// TIA Portal V15.1 export
// export: Created 2024-06-21T08:41:18.6949066Z, ExportSetting WithDefaults, DisplayName Totally Integrated Automation Portal, DisplayVersion V15.1 Update 5, DisplayName TIA Portal Openness, DisplayVersion V15.1 Update 5, DisplayName SINAMICS Startdrive Advanced, DisplayVersion V15.1, DisplayName G130, G150, S120, S150, SINAMICS MV, S210, DisplayVersion V15.1, DisplayName G110M, G120, G120C, G120D, G120P, DisplayVersion V15.1, DisplayName STEP 7 Professional, DisplayVersion V15.1 Update 5, DisplayName STEP 7 Safety, DisplayVersion V15.1, DisplayName WinCC Professional, DisplayVersion V15.1 Update 5, DisplayName SIMATIC Visualization Architect, DisplayVersion V15.1
FUNCTION_BLOCK "LGBLineConv-MDXPN-DFS22B"   // FB6682, FBD
TITLE = LGBLineConv-MDXPN-DFS22B
{ S7_Optimized_Access := 'TRUE' }
VERSION : 0.1
// stored: AutoNumber false, IsIECCheckEnabled false, IsRetainMemResEnabled false, MemoryReserve 100, SetENOAutomatically False, UDAEnableTagReadback false
   VAR_INPUT
      I_DetArrived { ExternalAccessible := 'False'; ExternalVisible := 'False'; ExternalWritable := 'False'} : Bool;   // Arrived detection
      I_DetSaturation { ExternalAccessible := 'False'; ExternalVisible := 'False'; ExternalWritable := 'False'} : Bool;   // Saturation detection
      I_DetMinGapLeft { ExternalAccessible := 'False'; ExternalVisible := 'False'; ExternalWritable := 'False'} : Bool;   // Minimum gap detection Left
      I_DetMinGapRight { ExternalAccessible := 'False'; ExternalVisible := 'False'; ExternalWritable := 'False'} : Bool;   // Minimum gap detection Right
      I_TrfInSetBegin { ExternalAccessible := 'False'; ExternalVisible := 'False'; ExternalWritable := 'False'} : Bool;   // Load Begin: condition to start transfer IN set
      I_TrfInSetIntlkOk { ExternalAccessible := 'False'; ExternalVisible := 'False'; ExternalWritable := 'False'} : Bool;   // Transfer IN Interlock Set OK
      I_TrfInSetRdyDlv { ExternalAccessible := 'False'; ExternalVisible := 'False'; ExternalWritable := 'False'} : Bool;   // Ready to deliver: Signal from previous object set
      I_TrfInSetTM { ExternalAccessible := 'False'; ExternalVisible := 'False'; ExternalWritable := 'False'} : Bool;   // Transfer busy signal from previous equipement set
      I_TrfOutSetBegin { ExternalAccessible := 'False'; ExternalVisible := 'False'; ExternalWritable := 'False'} : Bool;   // Unload Begin: condition to start transfer OUT set
      I_TrfOutSetIntlkOk { ExternalAccessible := 'False'; ExternalVisible := 'False'; ExternalWritable := 'False'} : Bool;   // Transfer Out Interlock Set Ok
      I_TrfOutSetRdyRcv { ExternalAccessible := 'False'; ExternalVisible := 'False'; ExternalWritable := 'False'} : Bool;   // Ready to Receive: Signal from next object set
      I_TrfOutSetArrived { ExternalAccessible := 'False'; ExternalVisible := 'False'; ExternalWritable := 'False'} : Bool;   // Body Arrived: Signal from next object Set
      I_StopProduction { ExternalAccessible := 'False'; ExternalVisible := 'False'; ExternalWritable := 'False'} : Bool;   // Stop Production
      I_ExtStopCondition { ExternalAccessible := 'False'; ExternalVisible := 'False'; ExternalWritable := 'False'} : Bool;   // External stop condition
      I_InfeedBegin { ExternalAccessible := 'False'; ExternalVisible := 'False'; ExternalWritable := 'False'} : Bool;   // Infeed begin
      I_ManInfeedAllowed { ExternalAccessible := 'False'; ExternalVisible := 'False'; ExternalWritable := 'False'} : Bool;   // Manual Infeed Allowed (without PushButton)
      I_EnabledriveCon { ExternalAccessible := 'False'; ExternalVisible := 'False'; ExternalWritable := 'False'} : Bool;   // Enable drive Condition
      I_MotorProtection { ExternalAccessible := 'False'; ExternalVisible := 'False'; ExternalWritable := 'False'} : Bool;   // Motorprotection
      I_BrakeProtection { ExternalAccessible := 'False'; ExternalVisible := 'False'; ExternalWritable := 'False'} : Bool;   // Brake protection
      I_SafetySwitch { ExternalAccessible := 'False'; ExternalVisible := 'False'; ExternalWritable := 'False'} : Bool;   // Safety switch
      I_LocalPBSet { ExternalAccessible := 'False'; ExternalVisible := 'False'; ExternalWritable := 'False'} : Bool;   // Push button for manual movememt (on local panel)
      I_LocalPBRes { ExternalAccessible := 'False'; ExternalVisible := 'False'; ExternalWritable := 'False'} : Bool;   // Push button for manual movememt Reset(on local panel)
      I_SafetyOk { ExternalAccessible := 'False'; ExternalVisible := 'False'; ExternalWritable := 'False'} : Bool := TRUE;   // Safety Ok
      I_MotionStopOk { ExternalAccessible := 'False'; ExternalVisible := 'False'; ExternalWritable := 'False'} : Bool;   // Safety Ok / The motion stop is Ok
      I_Speed { ExternalAccessible := 'False'; ExternalVisible := 'False'; ExternalWritable := 'False'} : Int;   // Speed Value in mm/s
      I_SafetyStatusWord1 { ExternalAccessible := 'False'; ExternalVisible := 'False'; ExternalWritable := 'False'} : Word;   // Safety Status Word
      I_SafetyStatusWord2 { ExternalAccessible := 'False'; ExternalVisible := 'False'; ExternalWritable := 'False'} : Word;   // Safety Status / Safety Status Word
      I_SafetyStatusWord3 { ExternalAccessible := 'False'; ExternalVisible := 'False'; ExternalWritable := 'False'} : Word;   // Safety Status / Safety Status Word
      I_SafetyControlWord1 { ExternalAccessible := 'False'; ExternalVisible := 'False'; ExternalWritable := 'False'} : Word;   // Safety Control Word
      I_SafetyControlWord2 { ExternalAccessible := 'False'; ExternalVisible := 'False'; ExternalWritable := 'False'} : Word;   // Safety Control Word
      I_SafetyControlWord3 { ExternalAccessible := 'False'; ExternalVisible := 'False'; ExternalWritable := 'False'} : Word;   // Safety Control Word
   END_VAR
   VAR_OUTPUT
      O_Active { ExternalAccessible := 'False'; ExternalVisible := 'False'; ExternalWritable := 'False'} : Bool;   // Is Active
      O_ReadyForOperation { ExternalAccessible := 'False'; ExternalVisible := 'False'; ExternalWritable := 'False'} : Bool;   // Ready for operation
      O_TrfInSetRdyRcv { ExternalAccessible := 'False'; ExternalVisible := 'False'; ExternalWritable := 'False'} : Bool;   // Ready to Receive: Signal to previous object set
      O_TrfInSetArrived { ExternalAccessible := 'False'; ExternalVisible := 'False'; ExternalWritable := 'False'} : Bool;   // Body Arrived: Signal to previous object Set
      O_TrfInSetActive { ExternalAccessible := 'False'; ExternalVisible := 'False'; ExternalWritable := 'False'} : Bool;   // Transfer in set active
      O_TrfInSetFinished { ExternalAccessible := 'False'; ExternalVisible := 'False'; ExternalWritable := 'False'} : Bool;   // Transfer in set finished
      O_TrfOutSetRdyDlv { ExternalAccessible := 'False'; ExternalVisible := 'False'; ExternalWritable := 'False'} : Bool;   // Ready to Deliver: Signal to next object set
      O_TrfOutSetTM { ExternalAccessible := 'False'; ExternalVisible := 'False'; ExternalWritable := 'False'} : Bool;   // Transfer: Signal to next object set
      O_TrfOutSetActive { ExternalAccessible := 'False'; ExternalVisible := 'False'; ExternalWritable := 'False'} : Bool;   // Transfer out set active
      O_TrfOutSetFinished { ExternalAccessible := 'False'; ExternalVisible := 'False'; ExternalWritable := 'False'} : Bool;   // Transfer out set finished
      O_Saturation { ExternalAccessible := 'False'; ExternalVisible := 'False'; ExternalWritable := 'False'} : Bool;   // Saturation
      O_EcoMode { ExternalAccessible := 'False'; ExternalVisible := 'False'; ExternalWritable := 'False'} : Bool;   // EcoMode is active
      O_EnableDrive { ExternalAccessible := 'False'; ExternalVisible := 'False'; ExternalWritable := 'False'} : Bool;   // Enable Drive
      O_LedRoller { ExternalAccessible := 'False'; ExternalVisible := 'False'; ExternalWritable := 'False'} : Bool;   // Led of roller
      O_AlarmABCondition { ExternalAccessible := 'False'; ExternalVisible := 'False'; ExternalWritable := 'False'} : Bool;   // Alarm AB condition
      O_AlarmA { ExternalAccessible := 'False'; ExternalVisible := 'False'; ExternalWritable := 'False'} : Bool;   // Alarm A
      O_AlarmB { ExternalAccessible := 'False'; ExternalVisible := 'False'; ExternalWritable := 'False'} : Bool;   // Alarm B
      O_AlarmC { ExternalAccessible := 'False'; ExternalVisible := 'False'; ExternalWritable := 'False'} : Bool;   // Alarm C
      O_AlarmD { ExternalAccessible := 'False'; ExternalVisible := 'False'; ExternalWritable := 'False'} : Bool;   // Alarm D
      H_AlarmWord { ExternalAccessible := 'False'; ExternalVisible := 'False'; ExternalWritable := 'False'} : DWord;   // Alarmword for WinCC
   END_VAR
   VAR_IN_OUT
      IO_Modes : "Modes";   // Modes
      H_HMI : "H_HMI";   // Animation
      "H_GBLineConv-MDXPN-DFS22B" : "H_GBLineConv-MDXPN-DFS22B";   // Animation
      C_Config : "LineConv-MDXPNConfig";   // Config
   END_VAR
   VAR
      AA_MotorProtection { ExternalAccessible := 'False'; ExternalVisible := 'False'; ExternalWritable := 'False'} : Bool;   // Motor Protection Tripped
      AA_BrakeProtection { ExternalAccessible := 'False'; ExternalVisible := 'False'; ExternalWritable := 'False'} : Bool;   // Brake Protection Tripped
      AA_SafetySwitch { ExternalAccessible := 'False'; ExternalVisible := 'False'; ExternalWritable := 'False'} : Bool;   // Safety Switch Not Ok
      AB_Alarm { ExternalAccessible := 'False'; ExternalVisible := 'False'; ExternalWritable := 'False'} : Bool;   // Frequency Control Alarm
      AB_MinGapLeft { ExternalAccessible := 'False'; ExternalVisible := 'False'; ExternalWritable := 'False'} : Bool;   // Minimum gap detection Left
      AB_MinGapRight { ExternalAccessible := 'False'; ExternalVisible := 'False'; ExternalWritable := 'False'} : Bool;   // Minimum gap detection Right
      AB_TrfOutSetOverTime { ExternalAccessible := 'False'; ExternalVisible := 'False'; ExternalWritable := 'False'} : Bool;   // Timeout Set
      AC_TrfInStopped { ExternalAccessible := 'False'; ExternalVisible := 'False'; ExternalWritable := 'False'} : Bool;   // Transfer In Stopped
      AC_MinGapLeft { ExternalAccessible := 'False'; ExternalVisible := 'False'; ExternalWritable := 'False'} : Bool;   // Minimum gap detection Left
      AC_MinGapRight { ExternalAccessible := 'False'; ExternalVisible := 'False'; ExternalWritable := 'False'} : Bool;   // Minimum gap detection Right
      AD_Warning { ExternalAccessible := 'False'; ExternalVisible := 'False'; ExternalWritable := 'False'} : Bool;   // Frequency Control Warning
      AD_TrfOutSetInterlock { ExternalAccessible := 'False'; ExternalVisible := 'False'; ExternalWritable := 'False'} : Bool;   // Interlock Not Ok Transport Out Set
      AD_TrfInSetInterlock { ExternalAccessible := 'False'; ExternalVisible := 'False'; ExternalWritable := 'False'} : Bool;   // Interlock Not Ok Transport In Set
      AD_SaturationState { ExternalAccessible := 'False'; ExternalVisible := 'False'; ExternalWritable := 'False'} : Bool;   // Saturation State
      AD_MotionStop { ExternalAccessible := 'False'; ExternalVisible := 'False'; ExternalWritable := 'False'} : Bool;   // Motion Stop
      AC_ConfigCalibrationAlm { ExternalAccessible := 'False'; ExternalVisible := 'False'; ExternalWritable := 'False'} : Bool;   // The Config values for Alarm Transfer time must be ALL zero or ALL different from zero
      AD_CalibrationSetWarn { ExternalAccessible := 'False'; ExternalVisible := 'False'; ExternalWritable := 'False'} : Bool;   // No High speed selected so Calibration is not possible for SET direction
      AC_ConfigRampAlm { ExternalAccessible := 'False'; ExternalVisible := 'False'; ExternalWritable := 'False'} : Bool;   // The config value for the ramp is not correct, must be zero or the config values for the calculation of the ramp must be ALL zero
      AC_ConfigRampCalcAlm { ExternalAccessible := 'False'; ExternalVisible := 'False'; ExternalWritable := 'False'} : Bool;   // The config values for the calculation of the ramp must be ALL different from zero
      SafetyOk { ExternalAccessible := 'False'; ExternalVisible := 'False'; ExternalWritable := 'False'} : Bool;   // Safety Ok
      TrfInfeedHoldSet { ExternalAccessible := 'False'; ExternalVisible := 'False'; ExternalWritable := 'False'} : Bool;   // Transfer infeed hold set driection
      TrfOutSetCmd { ExternalAccessible := 'False'; ExternalVisible := 'False'; ExternalWritable := 'False'} : Bool;   // Command after Interlock to Motor set
      TrfOutfeedHoldSet { ExternalAccessible := 'False'; ExternalVisible := 'False'; ExternalWritable := 'False'} : Bool;   // Transfer outfeed hold set direction
      TrfInSetCmd { ExternalAccessible := 'False'; ExternalVisible := 'False'; ExternalWritable := 'False'} : Bool;   // Command after Interlock to Motor set
      TrfInSetActive { ExternalAccessible := 'False'; ExternalVisible := 'False'; ExternalWritable := 'False'} : Bool;   // Load Active Set
      TrfOutSetActive { ExternalAccessible := 'False'; ExternalVisible := 'False'; ExternalWritable := 'False'} : Bool;   // Unload active Set
      TrfOutSetFinished { ExternalAccessible := 'False'; ExternalVisible := 'False'; ExternalWritable := 'False'} : Bool;   // Unload finished Set
      TrfOutSetRdyDlv { ExternalAccessible := 'False'; ExternalVisible := 'False'; ExternalWritable := 'False'} : Bool;   // Ready to Deliver: Signal to next object set
      TrfOutSetTM { ExternalAccessible := 'False'; ExternalVisible := 'False'; ExternalWritable := 'False'} : Bool;   // Transfer : Signal transfer memory to next object set
      TrfInSetRdyRcv { ExternalAccessible := 'False'; ExternalVisible := 'False'; ExternalWritable := 'False'} : Bool;   // Ready to Receive: Signal to previous object set
      TrfInSetArrived { ExternalAccessible := 'False'; ExternalVisible := 'False'; ExternalWritable := 'False'} : Bool;   // Body Arrived: Signal to previous object Set
      TrfInSetFinished { ExternalAccessible := 'False'; ExternalVisible := 'False'; ExternalWritable := 'False'} : Bool;   // Body Arrived: Signal to TrfOut module set (Reset TrfOutCmd)
      TrfOutSetAlmCond { ExternalAccessible := 'False'; ExternalVisible := 'False'; ExternalWritable := 'False'} : Bool;   // TrfOut Alarm condition
      TrfInSetTrfOutSetTM { ExternalAccessible := 'False'; ExternalVisible := 'False'; ExternalWritable := 'False'} : Bool;   // Transfer memory set
      MotorcmdHspdSet { ExternalAccessible := 'False'; ExternalVisible := 'False'; ExternalWritable := 'False'} : Bool;   // Command High Speed to Motorloop set
      MotorcmdHspdRes { ExternalAccessible := 'False'; ExternalVisible := 'False'; ExternalWritable := 'False'} : Bool;   // Command High Speed to Motorloop reset
      MotCmdAutoCond { ExternalAccessible := 'False'; ExternalVisible := 'False'; ExternalWritable := 'False'} : Bool;   // Motor Command Automatic Condition
      StationOnly { ExternalAccessible := 'False'; ExternalVisible := 'False'; ExternalWritable := 'False'} : Bool;   // Station only
      AlarmA { ExternalAccessible := 'False'; ExternalVisible := 'False'; ExternalWritable := 'False'} : Bool;   // Alarm A
      AlarmB { ExternalAccessible := 'False'; ExternalVisible := 'False'; ExternalWritable := 'False'} : Bool;   // Alarm B
      AlarmC { ExternalAccessible := 'False'; ExternalVisible := 'False'; ExternalWritable := 'False'} : Bool;   // Alarm C
      AlarmD { ExternalAccessible := 'False'; ExternalVisible := 'False'; ExternalWritable := 'False'} : Bool;   // Alarm D
      AlarmABCondition { ExternalAccessible := 'False'; ExternalVisible := 'False'; ExternalWritable := 'False'} : Bool;   // Alarm AB Condition
      MinGapLeftAlmCond { ExternalAccessible := 'False'; ExternalVisible := 'False'; ExternalWritable := 'False'} : Bool;   // Minimum gap detection Left Alarm condition
      MinGapRightAlmCond { ExternalAccessible := 'False'; ExternalVisible := 'False'; ExternalWritable := 'False'} : Bool;   // Minimum gap detection Right Alarm condition
      ReadyForOperation { ExternalAccessible := 'False'; ExternalVisible := 'False'; ExternalWritable := 'False'} : Bool;   // Ready for operation
      MotorLoopActive { ExternalAccessible := 'False'; ExternalVisible := 'False'; ExternalWritable := 'False'} : Bool;   // Motor Loop Active
      MotorLoopAlarmCond { ExternalAccessible := 'False'; ExternalVisible := 'False'; ExternalWritable := 'False'} : Bool;   // Motor loop Alarm condition
      PulsInfeedBegin { ExternalAccessible := 'False'; ExternalVisible := 'False'; ExternalWritable := 'False'} : Bool;   // Puls Infeed begin
      MaxTimeResetDirection { ExternalAccessible := 'False'; ExternalVisible := 'False'; ExternalWritable := 'False'} : Bool;   // Max Time Reset Direction
      LineConveyorEmpty { ExternalAccessible := 'False'; ExternalVisible := 'False'; ExternalWritable := 'False'} : Bool;   // Line conveyor is empty
      LineConveyorEmptyTime { ExternalAccessible := 'False'; ExternalVisible := 'False'; ExternalWritable := 'False'} : DInt;   // Time to empty Line conveyor (Msec)
      Edge { ExternalAccessible := 'False'; ExternalVisible := 'False'; ExternalWritable := 'False'} : Array[1..10] of Bool;   // Edge
      _LTrfInSet { ExternalAccessible := 'False'; ExternalVisible := 'False'; ExternalWritable := 'False'} : "LGBChainTrfIn";   // FB
      _LTrfOutSet { ExternalAccessible := 'False'; ExternalVisible := 'False'; ExternalWritable := 'False'} : "LGBTrfOut";   // FB
      _LineConv { ExternalAccessible := 'False'; ExternalVisible := 'False'; ExternalWritable := 'False'} : "LGBMotor2W2S-MDXPN-6PD-DFS22B";   // FB
      _CheckMinGapLeft { ExternalAccessible := 'False'; ExternalVisible := 'False'; ExternalWritable := 'False'} : "L1AlarmMultiIn";   // FB
      _CheckMinGapRight { ExternalAccessible := 'False'; ExternalVisible := 'False'; ExternalWritable := 'False'} : "L1AlarmMultiIn";   // FB
      _Check2MinGapLeft { ExternalAccessible := 'False'; ExternalVisible := 'False'; ExternalWritable := 'False'} : "L1AlarmMultiIn";   // FB
      _Check2MinGapRight { ExternalAccessible := 'False'; ExternalVisible := 'False'; ExternalWritable := 'False'} : "L1AlarmMultiIn";   // FB
      _StationOnly { ExternalAccessible := 'False'; ExternalVisible := 'False'; ExternalWritable := 'False'} : "LToggle";   // FB
      _NoTrfIn { ExternalAccessible := 'False'; ExternalVisible := 'False'; ExternalWritable := 'False'} : "LToggle";   // FB
      _Saturation { ExternalAccessible := 'False'; ExternalVisible := 'False'; ExternalWritable := 'False'} : IEC_TIMER;   // Timer
      _MaxTimeResetDirection { ExternalAccessible := 'False'; ExternalVisible := 'False'; ExternalWritable := 'False'} : IEC_TIMER;   // Timer
      _EcoMode { ExternalAccessible := 'False'; ExternalVisible := 'False'; ExternalWritable := 'False'} : IEC_TIMER;   // Timer
   END_VAR
   VAR_TEMP
      H_HMITrfInSet : "H_HMI";   // Temp
      H_HMITrfOutSet : "H_HMI";   // Temp
      H_HMIMotor : "H_HMI";   // Temp
      HMICMD : "ConvHMICMD";   // Temp
   END_VAR
   VAR_TEMP   // added for the SCL form of the ladder/FBD networks
      _w1 : Bool;
   END_VAR
BEGIN

REGION Network 1: **** 1 - Inputs **** HMI Commands
   // HMI Commands
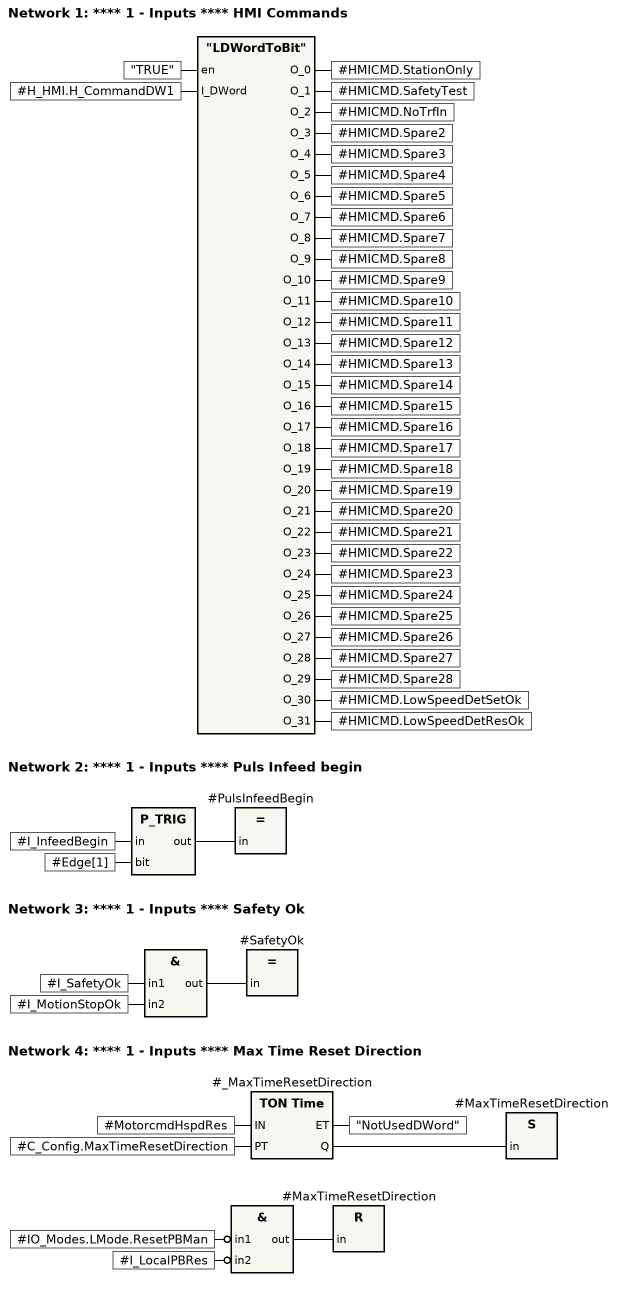
   IF "TRUE" THEN
       "LDWordToBit"(I_DWord := #H_HMI.H_CommandDW1,
                     O_0 => #HMICMD.StationOnly,
                     O_1 => #HMICMD.SafetyTest,
                     O_2 => #HMICMD.NoTrfIn,
                     O_3 => #HMICMD.Spare2,
                     O_4 => #HMICMD.Spare3,
                     O_5 => #HMICMD.Spare4,
                     O_6 => #HMICMD.Spare5,
                     O_7 => #HMICMD.Spare6,
                     O_8 => #HMICMD.Spare7,
                     O_9 => #HMICMD.Spare8,
                     O_10 => #HMICMD.Spare9,
                     O_11 => #HMICMD.Spare10,
                     O_12 => #HMICMD.Spare11,
                     O_13 => #HMICMD.Spare12,
                     O_14 => #HMICMD.Spare13,
                     O_15 => #HMICMD.Spare14,
                     O_16 => #HMICMD.Spare15,
                     O_17 => #HMICMD.Spare16,
                     O_18 => #HMICMD.Spare17,
                     O_19 => #HMICMD.Spare18,
                     O_20 => #HMICMD.Spare19,
                     O_21 => #HMICMD.Spare20,
                     O_22 => #HMICMD.Spare21,
                     O_23 => #HMICMD.Spare22,
                     O_24 => #HMICMD.Spare23,
                     O_25 => #HMICMD.Spare24,
                     O_26 => #HMICMD.Spare25,
                     O_27 => #HMICMD.Spare26,
                     O_28 => #HMICMD.Spare27,
                     O_29 => #HMICMD.Spare28,
                     O_30 => #HMICMD.LowSpeedDetSetOk,
                     O_31 => #HMICMD.LowSpeedDetResOk);
   END_IF;
END_REGION

REGION Network 2: **** 1 - Inputs **** Puls Infeed begin
   #_w1 := #I_InfeedBegin AND NOT #Edge[1];   // rising edge
   #Edge[1] := #I_InfeedBegin;
   #PulsInfeedBegin := #_w1;
END_REGION

REGION Network 3: **** 1 - Inputs **** Safety Ok
   #SafetyOk := #I_SafetyOk AND #I_MotionStopOk;
END_REGION

REGION Network 4: **** 1 - Inputs **** Max Time Reset Direction
   #_MaxTimeResetDirection.TON(IN := #MotorcmdHspdRes,
                           PT := #C_Config.MaxTimeResetDirection,
                           ET => "NotUsedDWord");
   IF #_MaxTimeResetDirection.Q THEN #MaxTimeResetDirection := TRUE; END_IF;
   IF NOT #IO_Modes.LMode.ResetPBMan AND NOT #I_LocalPBRes THEN #MaxTimeResetDirection := FALSE; END_IF;
END_REGION

REGION Network 5: **** 2.2 - Alarms - Alarms Generation **** AC-- Minimum gap detection Left
   // Alarm Minimum Gap1
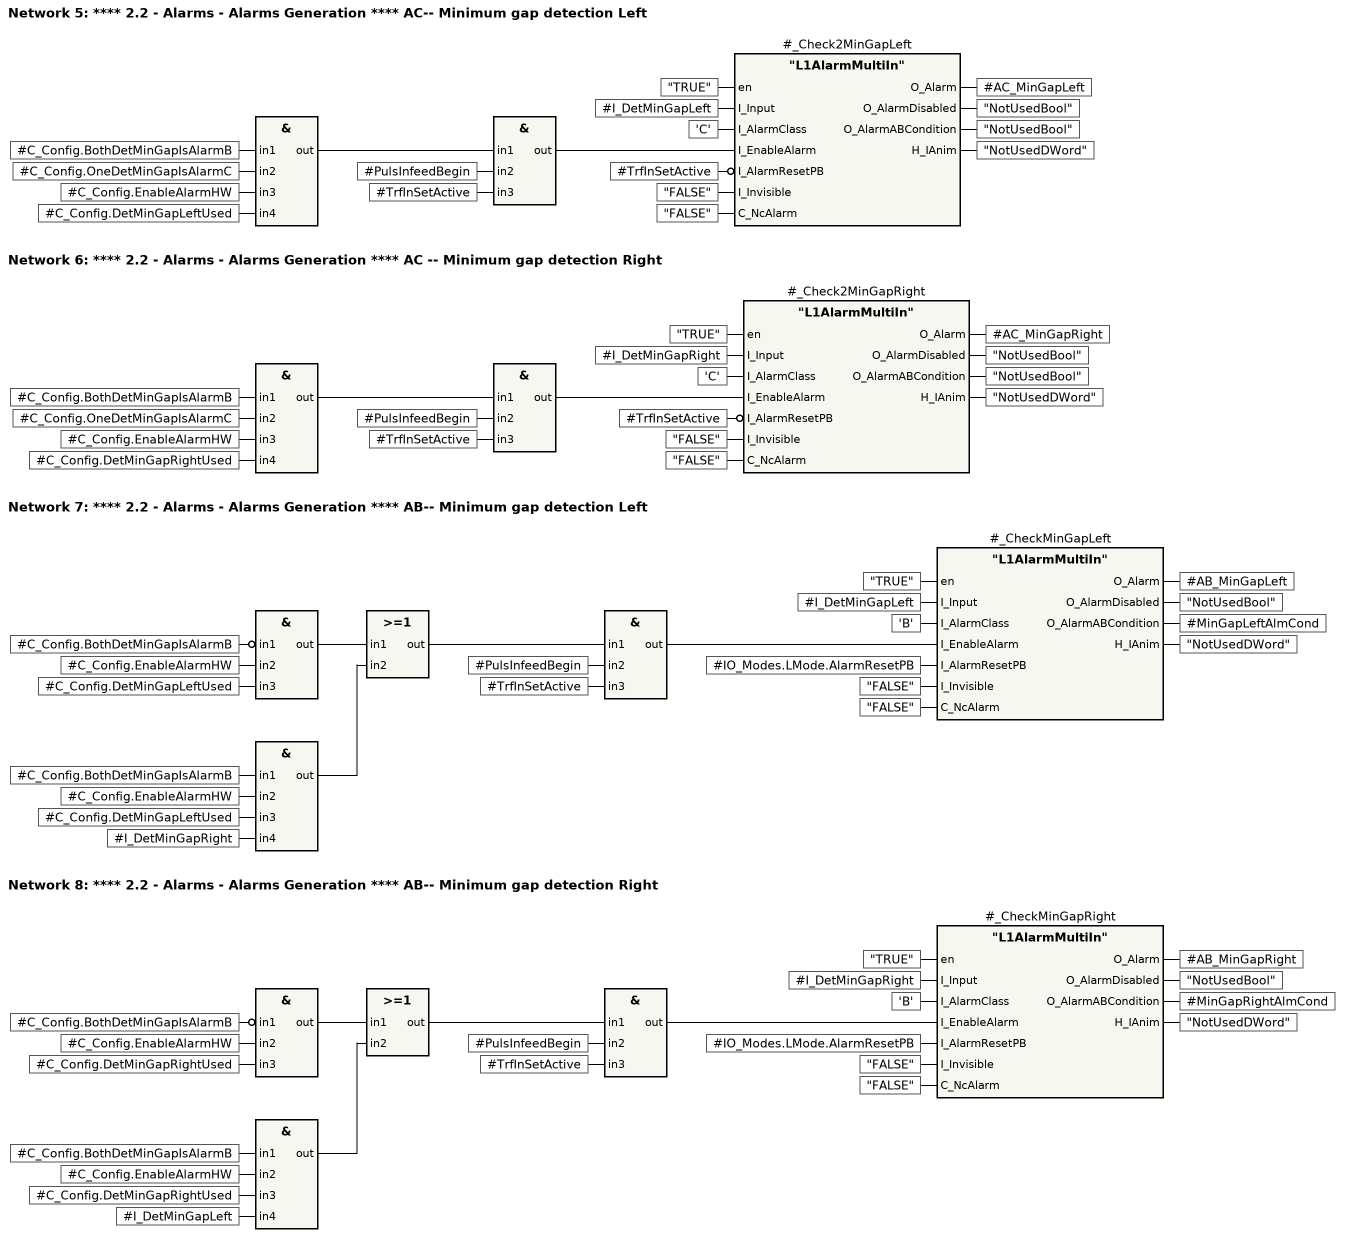
   IF "TRUE" THEN
       #_Check2MinGapLeft(I_Input := #I_DetMinGapLeft,   // "L1AlarmMultiIn"
                          I_AlarmClass := 'C',
                          I_EnableAlarm := #C_Config.BothDetMinGapIsAlarmB AND #C_Config.OneDetMinGapIsAlarmC AND #C_Config.EnableAlarmHW AND #C_Config.DetMinGapLeftUsed AND #PulsInfeedBegin AND #TrfInSetActive,
                          I_AlarmResetPB := NOT #TrfInSetActive,
                          I_Invisible := "FALSE",
                          C_NcAlarm := "FALSE",
                          O_Alarm => #AC_MinGapLeft,
                          O_AlarmDisabled => "NotUsedBool",
                          O_AlarmABCondition => "NotUsedBool",
                          H_IAnim => "NotUsedDWord");
   END_IF;
END_REGION

REGION Network 6: **** 2.2 - Alarms - Alarms Generation **** AC -- Minimum gap detection Right
   // Alarm Minimum Gap2
   IF "TRUE" THEN
       #_Check2MinGapRight(I_Input := #I_DetMinGapRight,   // "L1AlarmMultiIn"
                           I_AlarmClass := 'C',
                           I_EnableAlarm := #C_Config.BothDetMinGapIsAlarmB AND #C_Config.OneDetMinGapIsAlarmC AND #C_Config.EnableAlarmHW AND #C_Config.DetMinGapRightUsed AND #PulsInfeedBegin AND #TrfInSetActive,
                           I_AlarmResetPB := NOT #TrfInSetActive,
                           I_Invisible := "FALSE",
                           C_NcAlarm := "FALSE",
                           O_Alarm => #AC_MinGapRight,
                           O_AlarmDisabled => "NotUsedBool",
                           O_AlarmABCondition => "NotUsedBool",
                           H_IAnim => "NotUsedDWord");
   END_IF;
END_REGION

REGION Network 7: **** 2.2 - Alarms - Alarms Generation **** AB-- Minimum gap detection Left
   // Alarm Minimum Gap1
   IF "TRUE" THEN
       #_CheckMinGapLeft(I_Input := #I_DetMinGapLeft,   // "L1AlarmMultiIn"
                         I_AlarmClass := 'B',
                         I_EnableAlarm := ((NOT #C_Config.BothDetMinGapIsAlarmB AND #C_Config.EnableAlarmHW AND #C_Config.DetMinGapLeftUsed) OR (#C_Config.BothDetMinGapIsAlarmB AND #C_Config.EnableAlarmHW AND #C_Config.DetMinGapLeftUsed AND #I_DetMinGapRight)) AND #PulsInfeedBegin AND #TrfInSetActive,
                         I_AlarmResetPB := #IO_Modes.LMode.AlarmResetPB,
                         I_Invisible := "FALSE",
                         C_NcAlarm := "FALSE",
                         O_Alarm => #AB_MinGapLeft,
                         O_AlarmDisabled => "NotUsedBool",
                         O_AlarmABCondition => #MinGapLeftAlmCond,
                         H_IAnim => "NotUsedDWord");
   END_IF;
END_REGION

REGION Network 8: **** 2.2 - Alarms - Alarms Generation **** AB-- Minimum gap detection Right
   // Alarm Minimum Gap2
   IF "TRUE" THEN
       #_CheckMinGapRight(I_Input := #I_DetMinGapRight,   // "L1AlarmMultiIn"
                          I_AlarmClass := 'B',
                          I_EnableAlarm := ((NOT #C_Config.BothDetMinGapIsAlarmB AND #C_Config.EnableAlarmHW AND #C_Config.DetMinGapRightUsed) OR (#C_Config.BothDetMinGapIsAlarmB AND #C_Config.EnableAlarmHW AND #C_Config.DetMinGapRightUsed AND #I_DetMinGapLeft)) AND #PulsInfeedBegin AND #TrfInSetActive,
                          I_AlarmResetPB := #IO_Modes.LMode.AlarmResetPB,
                          I_Invisible := "FALSE",
                          C_NcAlarm := "FALSE",
                          O_Alarm => #AB_MinGapRight,
                          O_AlarmDisabled => "NotUsedBool",
                          O_AlarmABCondition => #MinGapRightAlmCond,
                          H_IAnim => "NotUsedDWord");
   END_IF;
END_REGION

REGION Network 9: **** 2.2 - Alarms - Alarms Generation **** Saturation Detection
   // Saturation Detection
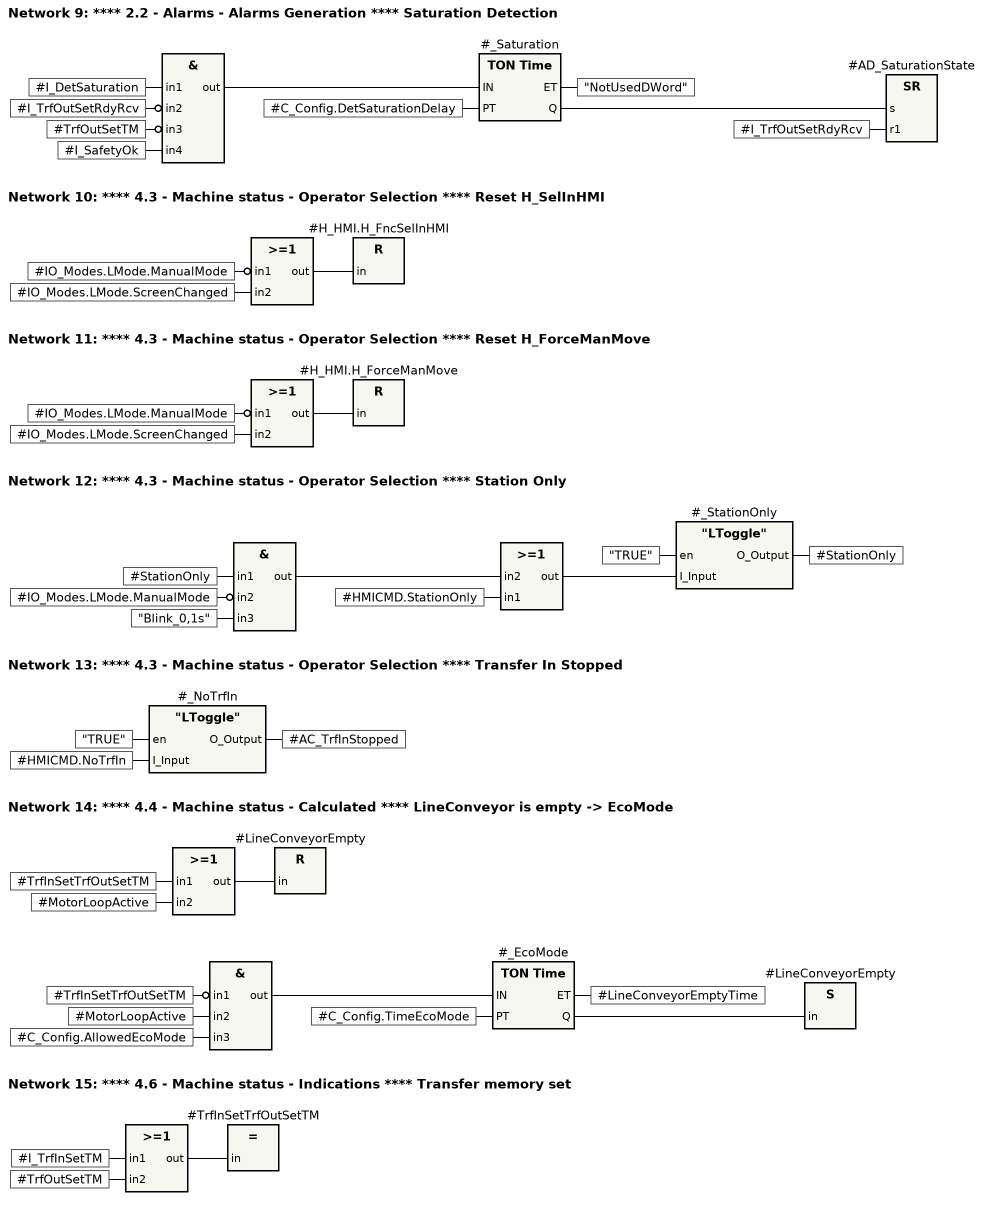
   #_Saturation.TON(IN := #I_DetSaturation AND NOT #I_TrfOutSetRdyRcv AND NOT #TrfOutSetTM AND #I_SafetyOk,
                    PT := #C_Config.DetSaturationDelay,
                    ET => "NotUsedDWord");
   IF #_Saturation.Q THEN
       #AD_SaturationState := TRUE;   // SR flip-flop
   END_IF;
   IF #I_TrfOutSetRdyRcv THEN #AD_SaturationState := FALSE; END_IF;
END_REGION

REGION Network 10: **** 4.3 - Machine status - Operator Selection **** Reset H_SelInHMI
   // Reset H_SelInHMI
   IF NOT #IO_Modes.LMode.ManualMode OR #IO_Modes.LMode.ScreenChanged THEN
       #H_HMI.H_FncSelInHMI := FALSE;
   END_IF;
END_REGION

REGION Network 11: **** 4.3 - Machine status - Operator Selection **** Reset H_ForceManMove
   // Reset H_ForceManMove
   IF NOT #IO_Modes.LMode.ManualMode OR #IO_Modes.LMode.ScreenChanged THEN
       #H_HMI.H_ForceManMove := FALSE;
   END_IF;
END_REGION

REGION Network 12: **** 4.3 - Machine status - Operator Selection **** Station Only
   // Station Only
   IF "TRUE" THEN
       #_StationOnly(I_Input := (#StationOnly AND NOT #IO_Modes.LMode.ManualMode AND "Blink_0,1s") OR #HMICMD.StationOnly,   // "LToggle"
                     O_Output => #StationOnly);
   END_IF;
END_REGION

REGION Network 13: **** 4.3 - Machine status - Operator Selection **** Transfer In Stopped
   // Transfer In Stopped
   IF "TRUE" THEN
       #_NoTrfIn(I_Input := #HMICMD.NoTrfIn, O_Output => #AC_TrfInStopped);   // "LToggle"
   END_IF;
END_REGION

REGION Network 14: **** 4.4 - Machine status - Calculated **** LineConveyor is empty -> EcoMode
   // LineConveyor is empty when chain is running and no detection is activated during the preset time
   IF #TrfInSetTrfOutSetTM OR #MotorLoopActive THEN #LineConveyorEmpty := FALSE; END_IF;
   #_EcoMode.TON(IN := NOT #TrfInSetTrfOutSetTM AND #MotorLoopActive AND #C_Config.AllowedEcoMode,
                 PT := #C_Config.TimeEcoMode,
                 ET => #LineConveyorEmptyTime);
   IF #_EcoMode.Q THEN #LineConveyorEmpty := TRUE; END_IF;
END_REGION

REGION Network 15: **** 4.6 - Machine status - Indications **** Transfer memory set
   // Transfer memory set
   #TrfInSetTrfOutSetTM := #I_TrfInSetTM OR #TrfOutSetTM;
END_REGION

REGION Network 16: **** 4.6 - Machine Status - Indication **** Icon Animation
   // Icon Animation
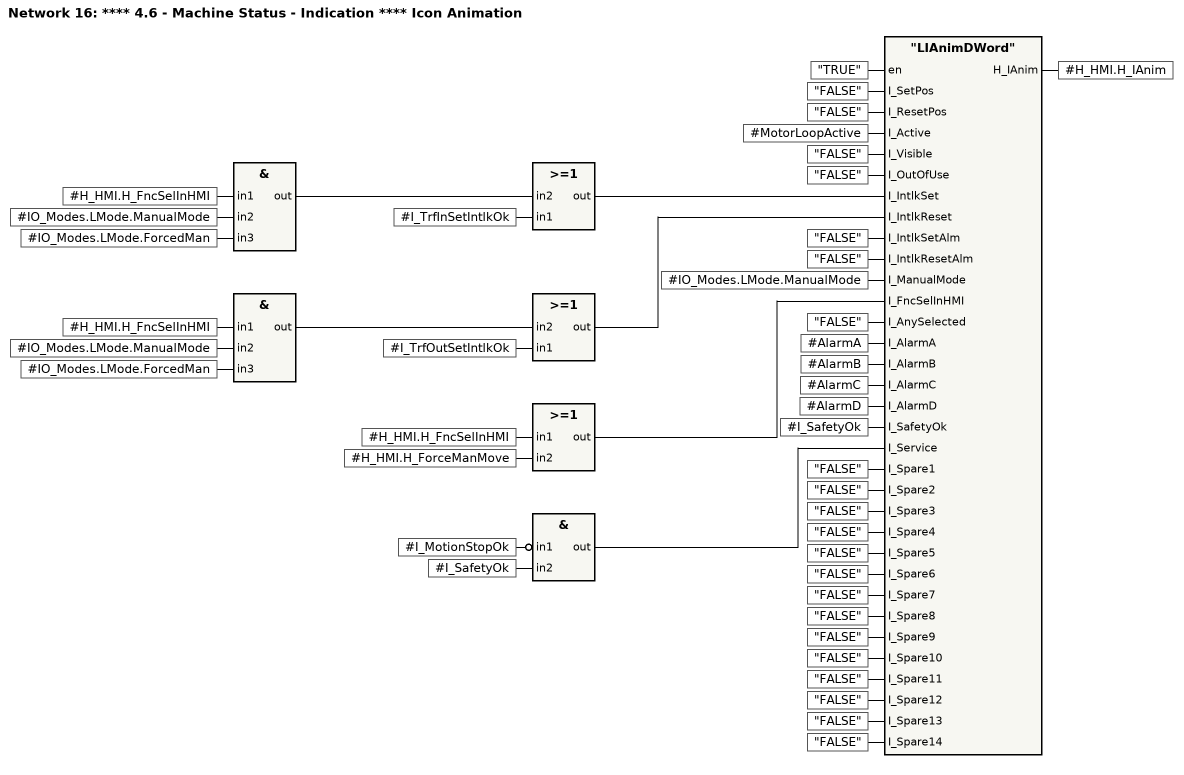
   IF "TRUE" THEN
       "LIAnimDWord"(I_SetPos := "FALSE",
                     I_ResetPos := "FALSE",
                     I_Active := #MotorLoopActive,
                     I_Visible := "FALSE",
                     I_OutOfUse := "FALSE",
                     I_IntlkSet := (#H_HMI.H_FncSelInHMI AND #IO_Modes.LMode.ManualMode AND #IO_Modes.LMode.ForcedMan) OR #I_TrfInSetIntlkOk,
                     I_IntlkReset := (#H_HMI.H_FncSelInHMI AND #IO_Modes.LMode.ManualMode AND #IO_Modes.LMode.ForcedMan) OR #I_TrfOutSetIntlkOk,
                     I_IntlkSetAlm := "FALSE",
                     I_IntlkResetAlm := "FALSE",
                     I_ManualMode := #IO_Modes.LMode.ManualMode,
                     I_FncSelInHMI := #H_HMI.H_FncSelInHMI OR #H_HMI.H_ForceManMove,
                     I_AnySelected := "FALSE",
                     I_AlarmA := #AlarmA,
                     I_AlarmB := #AlarmB,
                     I_AlarmC := #AlarmC,
                     I_AlarmD := #AlarmD,
                     I_SafetyOk := #I_SafetyOk,
                     I_Service := NOT #I_MotionStopOk AND #I_SafetyOk,
                     I_Spare1 := "FALSE",
                     I_Spare2 := "FALSE",
                     I_Spare3 := "FALSE",
                     I_Spare4 := "FALSE",
                     I_Spare5 := "FALSE",
                     I_Spare6 := "FALSE",
                     I_Spare7 := "FALSE",
                     I_Spare8 := "FALSE",
                     I_Spare9 := "FALSE",
                     I_Spare10 := "FALSE",
                     I_Spare11 := "FALSE",
                     I_Spare12 := "FALSE",
                     I_Spare13 := "FALSE",
                     I_Spare14 := "FALSE",
                     H_IAnim => #H_HMI.H_IAnim);
   END_IF;
END_REGION

REGION Network 17: **** 4.6 Machine status - Indications **** Arrived detection IAnim
   // Icon Animation
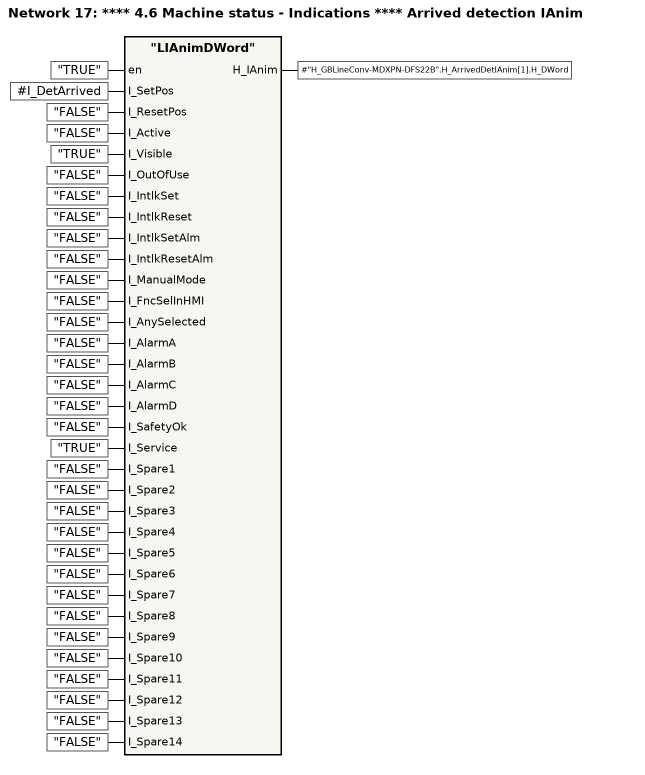
   IF "TRUE" THEN
       "LIAnimDWord"(I_SetPos := #I_DetArrived,
                     I_ResetPos := "FALSE",
                     I_Active := "FALSE",
                     I_Visible := "TRUE",
                     I_OutOfUse := "FALSE",
                     I_IntlkSet := "FALSE",
                     I_IntlkReset := "FALSE",
                     I_IntlkSetAlm := "FALSE",
                     I_IntlkResetAlm := "FALSE",
                     I_ManualMode := "FALSE",
                     I_FncSelInHMI := "FALSE",
                     I_AnySelected := "FALSE",
                     I_AlarmA := "FALSE",
                     I_AlarmB := "FALSE",
                     I_AlarmC := "FALSE",
                     I_AlarmD := "FALSE",
                     I_SafetyOk := "FALSE",
                     I_Service := "TRUE",
                     I_Spare1 := "FALSE",
                     I_Spare2 := "FALSE",
                     I_Spare3 := "FALSE",
                     I_Spare4 := "FALSE",
                     I_Spare5 := "FALSE",
                     I_Spare6 := "FALSE",
                     I_Spare7 := "FALSE",
                     I_Spare8 := "FALSE",
                     I_Spare9 := "FALSE",
                     I_Spare10 := "FALSE",
                     I_Spare11 := "FALSE",
                     I_Spare12 := "FALSE",
                     I_Spare13 := "FALSE",
                     I_Spare14 := "FALSE",
                     H_IAnim => #"H_GBLineConv-MDXPN-DFS22B".H_ArrivedDetIAnim[1].H_DWord);
   END_IF;
END_REGION

REGION Network 18: **** 4.6 Machine status - Indications **** Saturation detection IAnim
   // Icon Animation
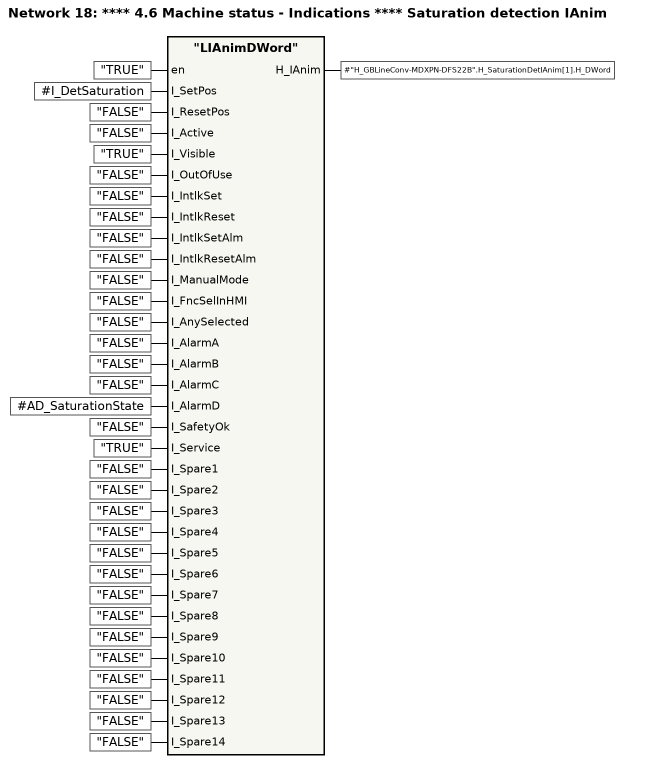
   IF "TRUE" THEN
       "LIAnimDWord"(I_SetPos := #I_DetSaturation,
                     I_ResetPos := "FALSE",
                     I_Active := "FALSE",
                     I_Visible := "TRUE",
                     I_OutOfUse := "FALSE",
                     I_IntlkSet := "FALSE",
                     I_IntlkReset := "FALSE",
                     I_IntlkSetAlm := "FALSE",
                     I_IntlkResetAlm := "FALSE",
                     I_ManualMode := "FALSE",
                     I_FncSelInHMI := "FALSE",
                     I_AnySelected := "FALSE",
                     I_AlarmA := "FALSE",
                     I_AlarmB := "FALSE",
                     I_AlarmC := "FALSE",
                     I_AlarmD := #AD_SaturationState,
                     I_SafetyOk := "FALSE",
                     I_Service := "TRUE",
                     I_Spare1 := "FALSE",
                     I_Spare2 := "FALSE",
                     I_Spare3 := "FALSE",
                     I_Spare4 := "FALSE",
                     I_Spare5 := "FALSE",
                     I_Spare6 := "FALSE",
                     I_Spare7 := "FALSE",
                     I_Spare8 := "FALSE",
                     I_Spare9 := "FALSE",
                     I_Spare10 := "FALSE",
                     I_Spare11 := "FALSE",
                     I_Spare12 := "FALSE",
                     I_Spare13 := "FALSE",
                     I_Spare14 := "FALSE",
                     H_IAnim => #"H_GBLineConv-MDXPN-DFS22B".H_SaturationDetIAnim[1].H_DWord);
   END_IF;
END_REGION

REGION Network 19: **** 4.6 Machine status - Indications **** Minimum gap detection Left IAnim
   // Icon Animation
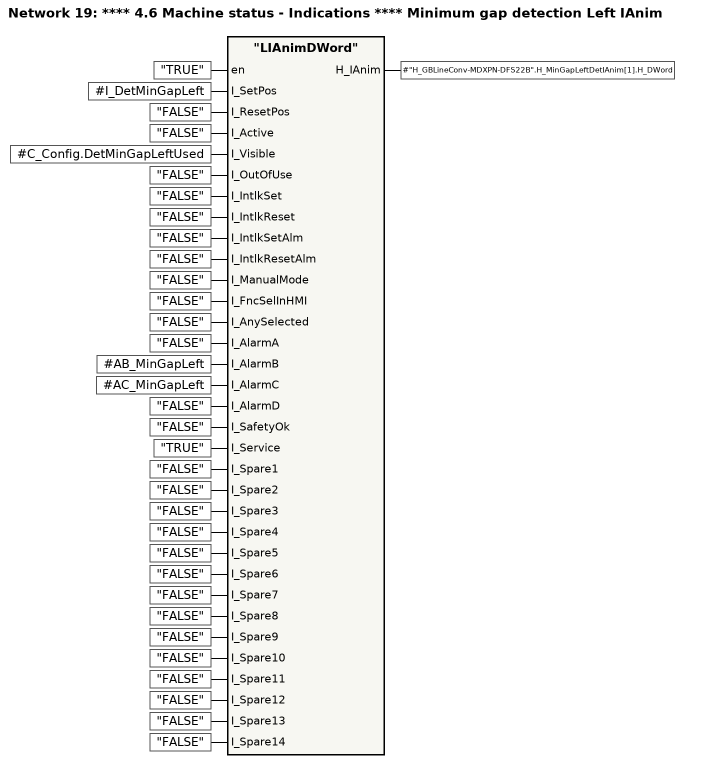
   IF "TRUE" THEN
       "LIAnimDWord"(I_SetPos := #I_DetMinGapLeft,
                     I_ResetPos := "FALSE",
                     I_Active := "FALSE",
                     I_Visible := #C_Config.DetMinGapLeftUsed,
                     I_OutOfUse := "FALSE",
                     I_IntlkSet := "FALSE",
                     I_IntlkReset := "FALSE",
                     I_IntlkSetAlm := "FALSE",
                     I_IntlkResetAlm := "FALSE",
                     I_ManualMode := "FALSE",
                     I_FncSelInHMI := "FALSE",
                     I_AnySelected := "FALSE",
                     I_AlarmA := "FALSE",
                     I_AlarmB := #AB_MinGapLeft,
                     I_AlarmC := #AC_MinGapLeft,
                     I_AlarmD := "FALSE",
                     I_SafetyOk := "FALSE",
                     I_Service := "TRUE",
                     I_Spare1 := "FALSE",
                     I_Spare2 := "FALSE",
                     I_Spare3 := "FALSE",
                     I_Spare4 := "FALSE",
                     I_Spare5 := "FALSE",
                     I_Spare6 := "FALSE",
                     I_Spare7 := "FALSE",
                     I_Spare8 := "FALSE",
                     I_Spare9 := "FALSE",
                     I_Spare10 := "FALSE",
                     I_Spare11 := "FALSE",
                     I_Spare12 := "FALSE",
                     I_Spare13 := "FALSE",
                     I_Spare14 := "FALSE",
                     H_IAnim => #"H_GBLineConv-MDXPN-DFS22B".H_MinGapLeftDetIAnim[1].H_DWord);
   END_IF;
END_REGION

REGION Network 20: **** 4.6 Machine status - Indications **** Minimum gap detection Right IAnim
   // Icon Animation
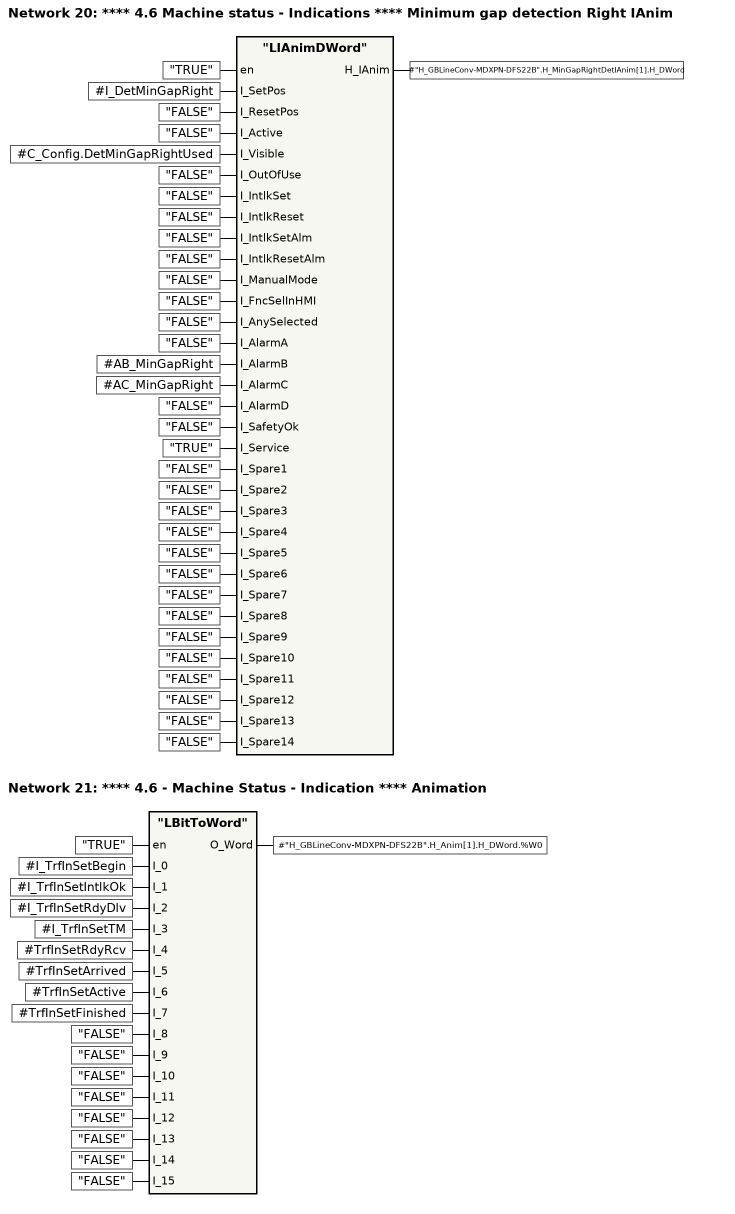
   IF "TRUE" THEN
       "LIAnimDWord"(I_SetPos := #I_DetMinGapRight,
                     I_ResetPos := "FALSE",
                     I_Active := "FALSE",
                     I_Visible := #C_Config.DetMinGapRightUsed,
                     I_OutOfUse := "FALSE",
                     I_IntlkSet := "FALSE",
                     I_IntlkReset := "FALSE",
                     I_IntlkSetAlm := "FALSE",
                     I_IntlkResetAlm := "FALSE",
                     I_ManualMode := "FALSE",
                     I_FncSelInHMI := "FALSE",
                     I_AnySelected := "FALSE",
                     I_AlarmA := "FALSE",
                     I_AlarmB := #AB_MinGapRight,
                     I_AlarmC := #AC_MinGapRight,
                     I_AlarmD := "FALSE",
                     I_SafetyOk := "FALSE",
                     I_Service := "TRUE",
                     I_Spare1 := "FALSE",
                     I_Spare2 := "FALSE",
                     I_Spare3 := "FALSE",
                     I_Spare4 := "FALSE",
                     I_Spare5 := "FALSE",
                     I_Spare6 := "FALSE",
                     I_Spare7 := "FALSE",
                     I_Spare8 := "FALSE",
                     I_Spare9 := "FALSE",
                     I_Spare10 := "FALSE",
                     I_Spare11 := "FALSE",
                     I_Spare12 := "FALSE",
                     I_Spare13 := "FALSE",
                     I_Spare14 := "FALSE",
                     H_IAnim => #"H_GBLineConv-MDXPN-DFS22B".H_MinGapRightDetIAnim[1].H_DWord);
   END_IF;
END_REGION

REGION Network 21: **** 4.6 - Machine Status - Indication **** Animation
   // Animation
   IF "TRUE" THEN
       "LBitToWord"(I_0 := #I_TrfInSetBegin,
                    I_1 := #I_TrfInSetIntlkOk,
                    I_2 := #I_TrfInSetRdyDlv,
                    I_3 := #I_TrfInSetTM,
                    I_4 := #TrfInSetRdyRcv,
                    I_5 := #TrfInSetArrived,
                    I_6 := #TrfInSetActive,
                    I_7 := #TrfInSetFinished,
                    I_8 := "FALSE",
                    I_9 := "FALSE",
                    I_10 := "FALSE",
                    I_11 := "FALSE",
                    I_12 := "FALSE",
                    I_13 := "FALSE",
                    I_14 := "FALSE",
                    I_15 := "FALSE",
                    O_Word => #"H_GBLineConv-MDXPN-DFS22B".H_Anim[1].H_DWord.%W0);
   END_IF;
END_REGION

REGION Network 22: **** 4.6 - Machine Status - Indication **** Animation
   // Animation
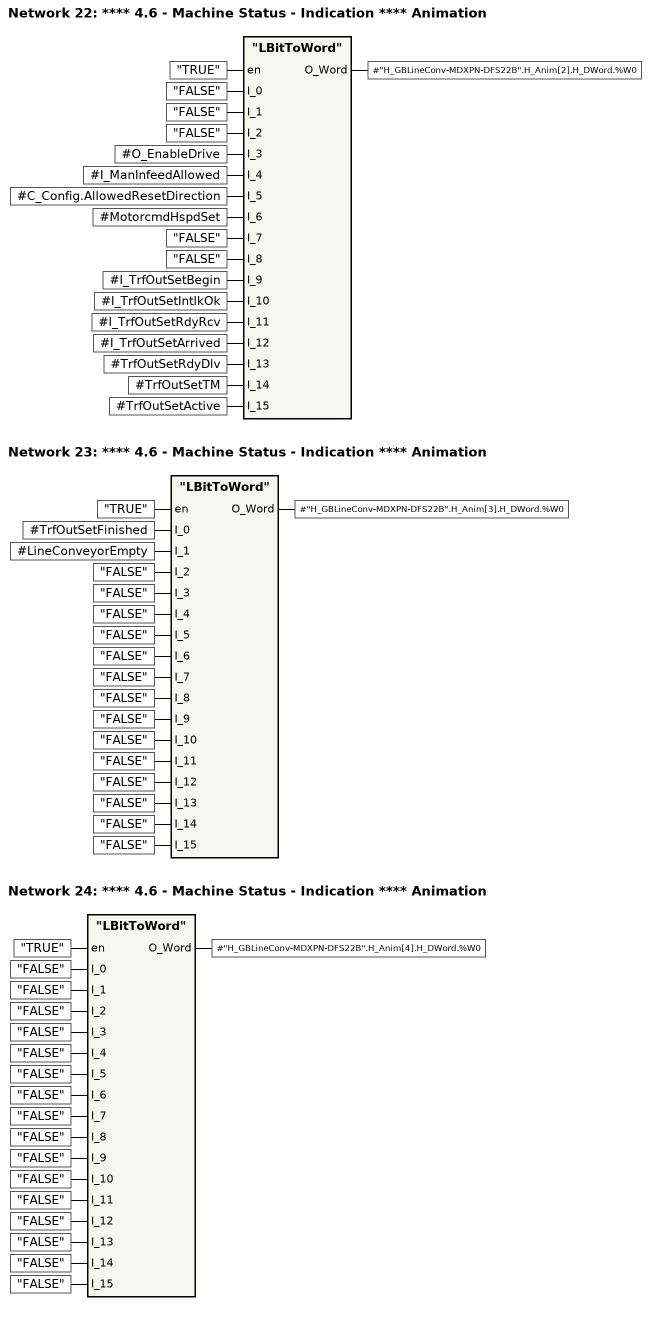
   IF "TRUE" THEN
       "LBitToWord"(I_0 := "FALSE",
                    I_1 := "FALSE",
                    I_2 := "FALSE",
                    I_3 := #O_EnableDrive,
                    I_4 := #I_ManInfeedAllowed,
                    I_5 := #C_Config.AllowedResetDirection,
                    I_6 := #MotorcmdHspdSet,
                    I_7 := "FALSE",
                    I_8 := "FALSE",
                    I_9 := #I_TrfOutSetBegin,
                    I_10 := #I_TrfOutSetIntlkOk,
                    I_11 := #I_TrfOutSetRdyRcv,
                    I_12 := #I_TrfOutSetArrived,
                    I_13 := #TrfOutSetRdyDlv,
                    I_14 := #TrfOutSetTM,
                    I_15 := #TrfOutSetActive,
                    O_Word => #"H_GBLineConv-MDXPN-DFS22B".H_Anim[2].H_DWord.%W0);
   END_IF;
END_REGION

REGION Network 23: **** 4.6 - Machine Status - Indication **** Animation
   // Animation
   IF "TRUE" THEN
       "LBitToWord"(I_0 := #TrfOutSetFinished,
                    I_1 := #LineConveyorEmpty,
                    I_2 := "FALSE",
                    I_3 := "FALSE",
                    I_4 := "FALSE",
                    I_5 := "FALSE",
                    I_6 := "FALSE",
                    I_7 := "FALSE",
                    I_8 := "FALSE",
                    I_9 := "FALSE",
                    I_10 := "FALSE",
                    I_11 := "FALSE",
                    I_12 := "FALSE",
                    I_13 := "FALSE",
                    I_14 := "FALSE",
                    I_15 := "FALSE",
                    O_Word => #"H_GBLineConv-MDXPN-DFS22B".H_Anim[3].H_DWord.%W0);
   END_IF;
END_REGION

REGION Network 24: **** 4.6 - Machine Status - Indication **** Animation
   // Animation
   IF "TRUE" THEN
       "LBitToWord"(I_0 := "FALSE",
                    I_1 := "FALSE",
                    I_2 := "FALSE",
                    I_3 := "FALSE",
                    I_4 := "FALSE",
                    I_5 := "FALSE",
                    I_6 := "FALSE",
                    I_7 := "FALSE",
                    I_8 := "FALSE",
                    I_9 := "FALSE",
                    I_10 := "FALSE",
                    I_11 := "FALSE",
                    I_12 := "FALSE",
                    I_13 := "FALSE",
                    I_14 := "FALSE",
                    I_15 := "FALSE",
                    O_Word => #"H_GBLineConv-MDXPN-DFS22B".H_Anim[4].H_DWord.%W0);
   END_IF;
END_REGION

REGION Network 25: **** 4.6 - Machine status - Indications **** Animation Time Chain Stop
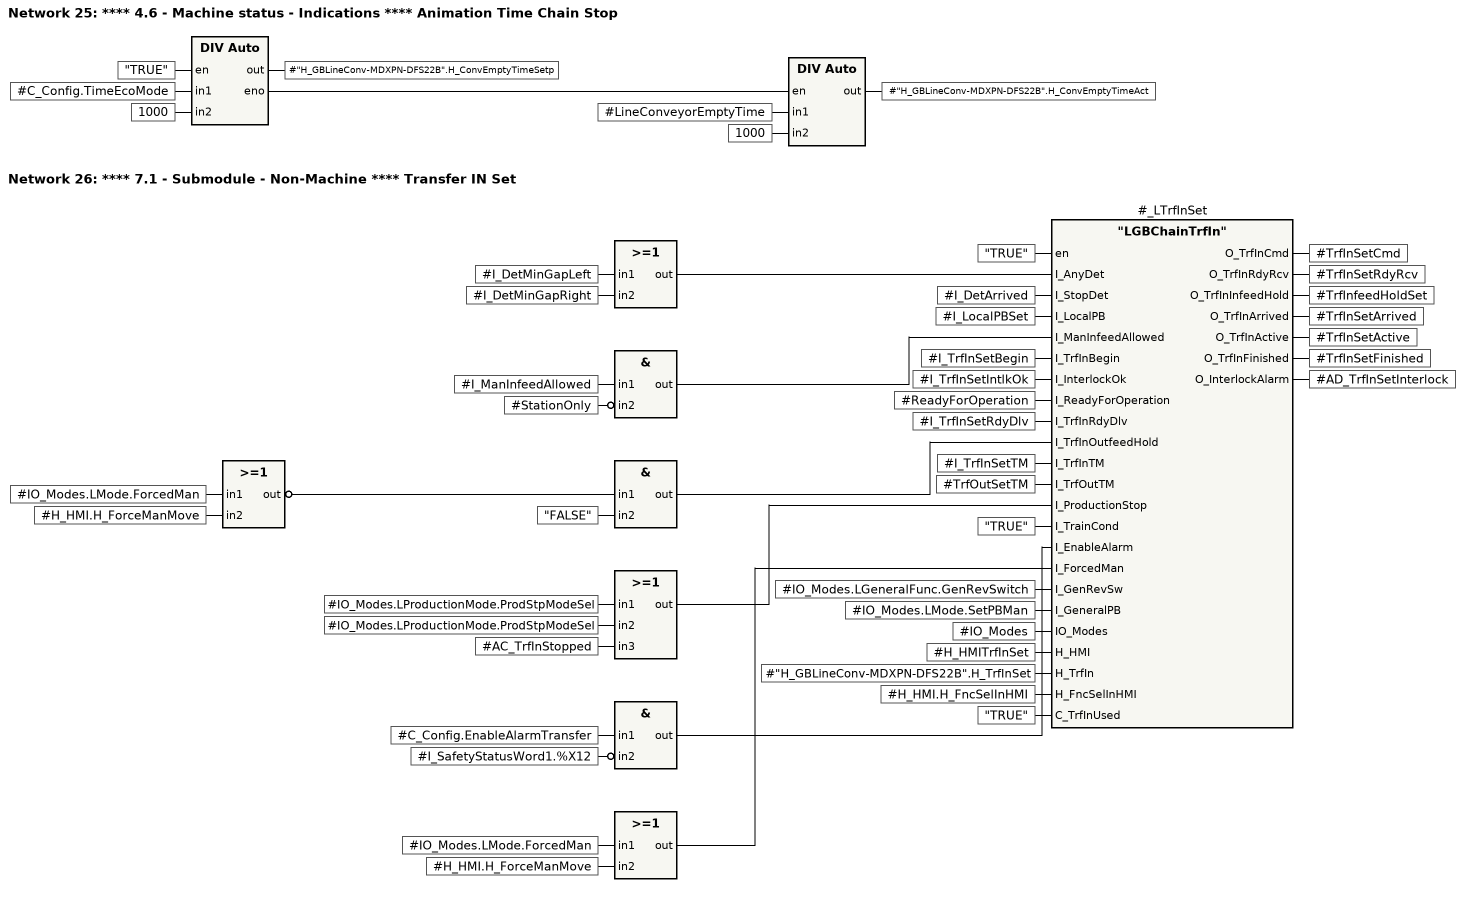
   IF "TRUE" THEN
       #"H_GBLineConv-MDXPN-DFS22B".H_ConvEmptyTimeSetp := #C_Config.TimeEcoMode / 1000;
       #"H_GBLineConv-MDXPN-DFS22B".H_ConvEmptyTimeAct := #LineConveyorEmptyTime / 1000;
   END_IF;
END_REGION

REGION Network 26: **** 7.1 - Submodule - Non-Machine **** Transfer IN Set
   // Transfer IN Set
   IF "TRUE" THEN
       #_LTrfInSet(I_AnyDet := #I_DetMinGapLeft OR #I_DetMinGapRight,   // "LGBChainTrfIn"
                   I_StopDet := #I_DetArrived,
                   I_LocalPB := #I_LocalPBSet,
                   I_ManInfeedAllowed := #I_ManInfeedAllowed AND NOT #StationOnly,
                   I_TrfInBegin := #I_TrfInSetBegin,
                   I_InterlockOk := #I_TrfInSetIntlkOk,
                   I_ReadyForOperation := #ReadyForOperation,
                   I_TrfInRdyDlv := #I_TrfInSetRdyDlv,
                   I_TrfInOutfeedHold := NOT (#IO_Modes.LMode.ForcedMan OR #H_HMI.H_ForceManMove) AND "FALSE",
                   I_TrfInTM := #I_TrfInSetTM,
                   I_TrfOutTM := #TrfOutSetTM,
                   I_ProductionStop := #IO_Modes.LProductionMode.ProdStpModeSel OR #IO_Modes.LProductionMode.ProdStpModeSel OR #AC_TrfInStopped,
                   I_TrainCond := "TRUE",
                   I_EnableAlarm := #C_Config.EnableAlarmTransfer AND NOT #I_SafetyStatusWord1.%X12,
                   I_ForcedMan := #IO_Modes.LMode.ForcedMan OR #H_HMI.H_ForceManMove,
                   I_GenRevSw := #IO_Modes.LGeneralFunc.GenRevSwitch,
                   I_GeneralPB := #IO_Modes.LMode.SetPBMan,
                   IO_Modes := #IO_Modes,
                   H_HMI := #H_HMITrfInSet,
                   H_TrfIn := #"H_GBLineConv-MDXPN-DFS22B".H_TrfInSet,
                   H_FncSelInHMI := #H_HMI.H_FncSelInHMI,
                   C_TrfInUsed := "TRUE",
                   O_TrfInCmd => #TrfInSetCmd,
                   O_TrfInRdyRcv => #TrfInSetRdyRcv,
                   O_TrfInInfeedHold => #TrfInfeedHoldSet,
                   O_TrfInArrived => #TrfInSetArrived,
                   O_TrfInActive => #TrfInSetActive,
                   O_TrfInFinished => #TrfInSetFinished,
                   O_InterlockAlarm => #AD_TrfInSetInterlock);
   END_IF;
END_REGION

REGION Network 27: **** 7.1 - Submodule - Non-Machine **** Transfer Out Set
   // Transfer Out Set
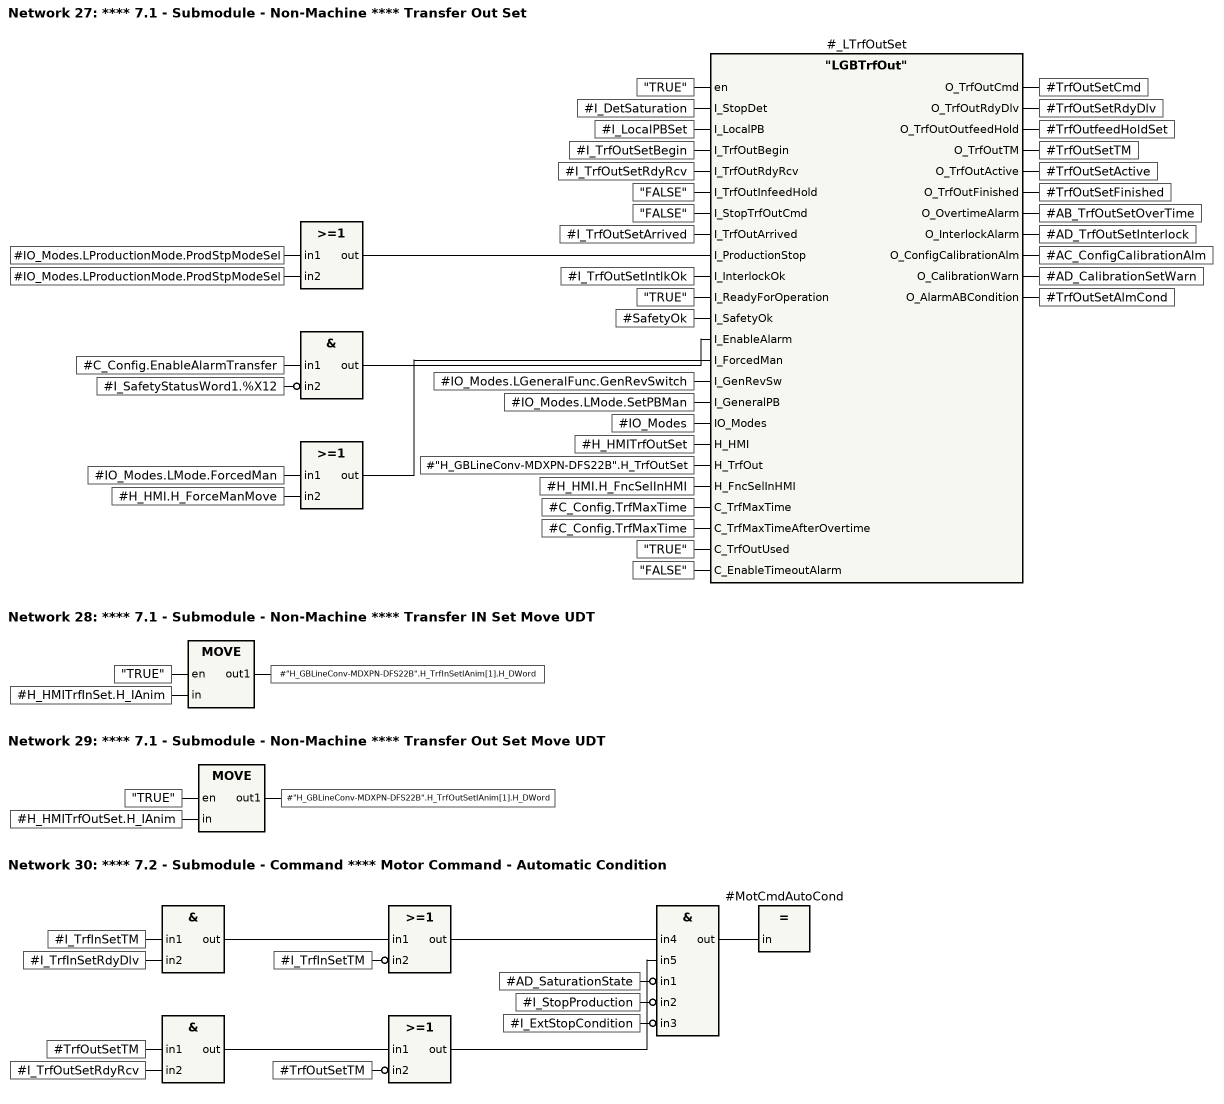
   IF "TRUE" THEN
       #_LTrfOutSet(I_StopDet := #I_DetSaturation,   // "LGBTrfOut"
                    I_LocalPB := #I_LocalPBSet,
                    I_TrfOutBegin := #I_TrfOutSetBegin,
                    I_TrfOutRdyRcv := #I_TrfOutSetRdyRcv,
                    I_TrfOutInfeedHold := "FALSE",
                    I_StopTrfOutCmd := "FALSE",
                    I_TrfOutArrived := #I_TrfOutSetArrived,
                    I_ProductionStop := #IO_Modes.LProductionMode.ProdStpModeSel OR #IO_Modes.LProductionMode.ProdStpModeSel,
                    I_InterlockOk := #I_TrfOutSetIntlkOk,
                    I_ReadyForOperation := "TRUE",
                    I_SafetyOk := #SafetyOk,
                    I_EnableAlarm := #C_Config.EnableAlarmTransfer AND NOT #I_SafetyStatusWord1.%X12,
                    I_ForcedMan := #IO_Modes.LMode.ForcedMan OR #H_HMI.H_ForceManMove,
                    I_GenRevSw := #IO_Modes.LGeneralFunc.GenRevSwitch,
                    I_GeneralPB := #IO_Modes.LMode.SetPBMan,
                    IO_Modes := #IO_Modes,
                    H_HMI := #H_HMITrfOutSet,
                    H_TrfOut := #"H_GBLineConv-MDXPN-DFS22B".H_TrfOutSet,
                    H_FncSelInHMI := #H_HMI.H_FncSelInHMI,
                    C_TrfMaxTime := #C_Config.TrfMaxTime,
                    C_TrfMaxTimeAfterOvertime := #C_Config.TrfMaxTime,
                    C_TrfOutUsed := "TRUE",
                    C_EnableTimeoutAlarm := "FALSE",
                    O_TrfOutCmd => #TrfOutSetCmd,
                    O_TrfOutRdyDlv => #TrfOutSetRdyDlv,
                    O_TrfOutOutfeedHold => #TrfOutfeedHoldSet,
                    O_TrfOutTM => #TrfOutSetTM,
                    O_TrfOutActive => #TrfOutSetActive,
                    O_TrfOutFinished => #TrfOutSetFinished,
                    O_OvertimeAlarm => #AB_TrfOutSetOverTime,
                    O_InterlockAlarm => #AD_TrfOutSetInterlock,
                    O_ConfigCalibrationAlm => #AC_ConfigCalibrationAlm,
                    O_CalibrationWarn => #AD_CalibrationSetWarn,
                    O_AlarmABCondition => #TrfOutSetAlmCond);
   END_IF;
END_REGION

REGION Network 28: **** 7.1 - Submodule - Non-Machine **** Transfer IN Set Move UDT
   // Transfer IN Set Move UDT
   IF "TRUE" THEN #"H_GBLineConv-MDXPN-DFS22B".H_TrfInSetIAnim[1].H_DWord := #H_HMITrfInSet.H_IAnim; END_IF;
END_REGION

REGION Network 29: **** 7.1 - Submodule - Non-Machine **** Transfer Out Set Move UDT
   // Transfer Out Set Move UDT
   IF "TRUE" THEN
       #"H_GBLineConv-MDXPN-DFS22B".H_TrfOutSetIAnim[1].H_DWord := #H_HMITrfOutSet.H_IAnim;
   END_IF;
END_REGION

REGION Network 30: **** 7.2 - Submodule - Command **** Motor Command - Automatic Condition
   #MotCmdAutoCond := ((#I_TrfInSetTM AND #I_TrfInSetRdyDlv) OR NOT #I_TrfInSetTM) AND ((#TrfOutSetTM AND #I_TrfOutSetRdyRcv) OR NOT #TrfOutSetTM) AND NOT #AD_SaturationState AND NOT #I_StopProduction AND NOT #I_ExtStopCondition;
END_REGION

REGION Network 31: **** 7.2 - Submodule - Command Summary **** Motor Command high speed Set
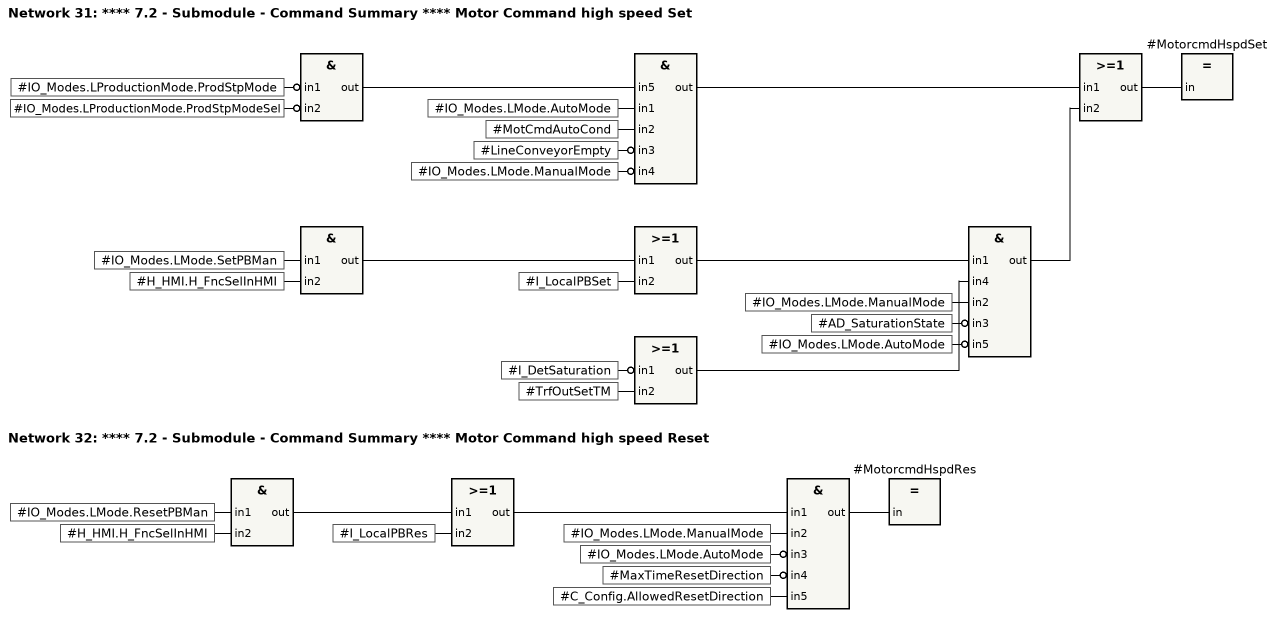
   #MotorcmdHspdSet := (NOT #IO_Modes.LProductionMode.ProdStpMode AND NOT #IO_Modes.LProductionMode.ProdStpModeSel AND #IO_Modes.LMode.AutoMode AND #MotCmdAutoCond AND NOT #LineConveyorEmpty AND NOT #IO_Modes.LMode.ManualMode) OR (((#IO_Modes.LMode.SetPBMan AND #H_HMI.H_FncSelInHMI) OR #I_LocalPBSet) AND (NOT #I_DetSaturation OR #TrfOutSetTM) AND #IO_Modes.LMode.ManualMode AND NOT #AD_SaturationState AND NOT #IO_Modes.LMode.AutoMode);
END_REGION

REGION Network 32: **** 7.2 - Submodule - Command Summary **** Motor Command high speed Reset
   #MotorcmdHspdRes := ((#IO_Modes.LMode.ResetPBMan AND #H_HMI.H_FncSelInHMI) OR #I_LocalPBRes) AND #IO_Modes.LMode.ManualMode AND NOT #IO_Modes.LMode.AutoMode AND NOT #MaxTimeResetDirection AND #C_Config.AllowedResetDirection;
END_REGION

REGION Network 33: **** 7.3 - Submodule - Machine **** Motor loop MoviDrive
   // Motor loop
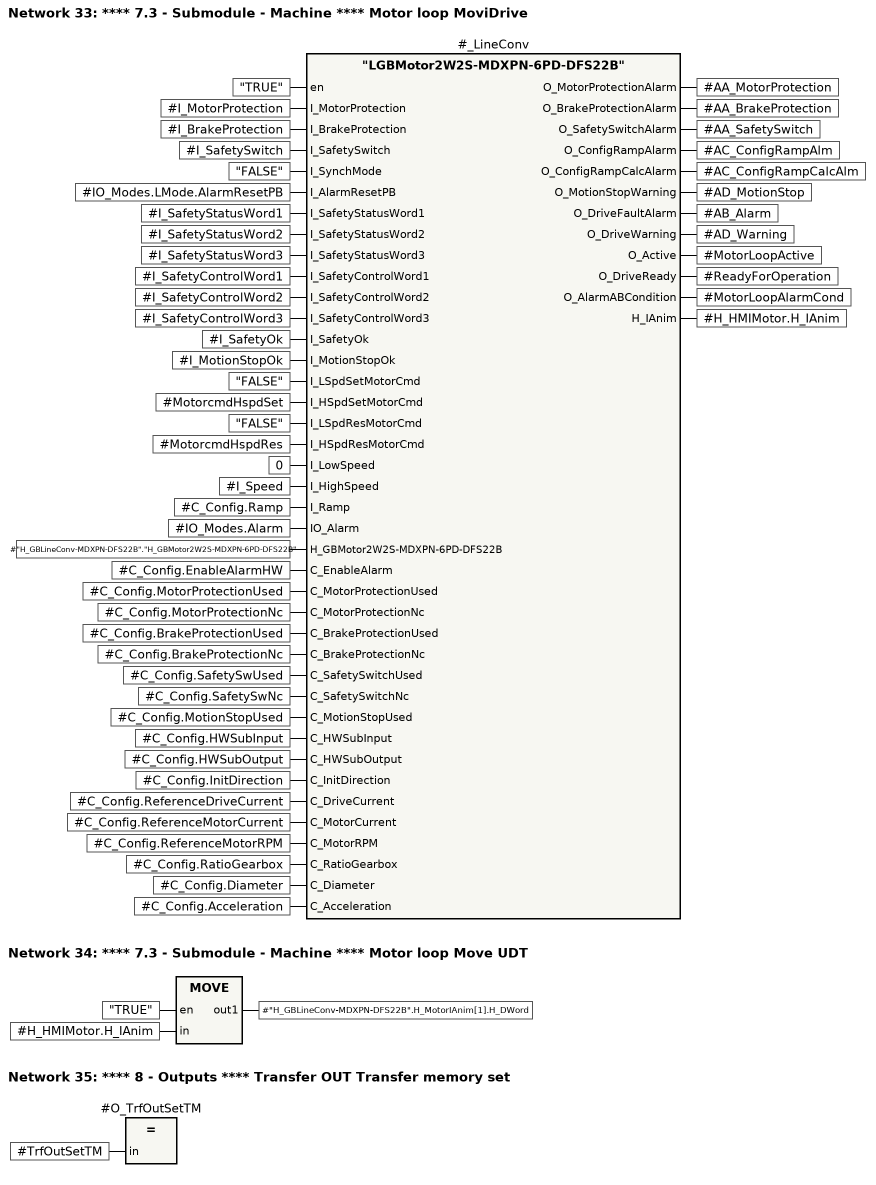
   IF "TRUE" THEN
       #_LineConv(I_MotorProtection := #I_MotorProtection,   // "LGBMotor2W2S-MDXPN-6PD-DFS22B"
                  I_BrakeProtection := #I_BrakeProtection,
                  I_SafetySwitch := #I_SafetySwitch,
                  I_SynchMode := "FALSE",
                  I_AlarmResetPB := #IO_Modes.LMode.AlarmResetPB,
                  I_SafetyStatusWord1 := #I_SafetyStatusWord1,
                  I_SafetyStatusWord2 := #I_SafetyStatusWord2,
                  I_SafetyStatusWord3 := #I_SafetyStatusWord3,
                  I_SafetyControlWord1 := #I_SafetyControlWord1,
                  I_SafetyControlWord2 := #I_SafetyControlWord2,
                  I_SafetyControlWord3 := #I_SafetyControlWord3,
                  I_SafetyOk := #I_SafetyOk,
                  I_MotionStopOk := #I_MotionStopOk,
                  I_LSpdSetMotorCmd := "FALSE",
                  I_HSpdSetMotorCmd := #MotorcmdHspdSet,
                  I_LSpdResMotorCmd := "FALSE",
                  I_HSpdResMotorCmd := #MotorcmdHspdRes,
                  I_LowSpeed := 0,
                  I_HighSpeed := #I_Speed,
                  I_Ramp := #C_Config.Ramp,
                  IO_Alarm := #IO_Modes.Alarm,
                  "H_GBMotor2W2S-MDXPN-6PD-DFS22B" := #"H_GBLineConv-MDXPN-DFS22B"."H_GBMotor2W2S-MDXPN-6PD-DFS22B",
                  C_EnableAlarm := #C_Config.EnableAlarmHW,
                  C_MotorProtectionUsed := #C_Config.MotorProtectionUsed,
                  C_MotorProtectionNc := #C_Config.MotorProtectionNc,
                  C_BrakeProtectionUsed := #C_Config.BrakeProtectionUsed,
                  C_BrakeProtectionNc := #C_Config.BrakeProtectionNc,
                  C_SafetySwitchUsed := #C_Config.SafetySwUsed,
                  C_SafetySwitchNc := #C_Config.SafetySwNc,
                  C_MotionStopUsed := #C_Config.MotionStopUsed,
                  C_HWSubInput := #C_Config.HWSubInput,
                  C_HWSubOutput := #C_Config.HWSubOutput,
                  C_InitDirection := #C_Config.InitDirection,
                  C_DriveCurrent := #C_Config.ReferenceDriveCurrent,
                  C_MotorCurrent := #C_Config.ReferenceMotorCurrent,
                  C_MotorRPM := #C_Config.ReferenceMotorRPM,
                  C_RatioGearbox := #C_Config.RatioGearbox,
                  C_Diameter := #C_Config.Diameter,
                  C_Acceleration := #C_Config.Acceleration,
                  O_MotorProtectionAlarm => #AA_MotorProtection,
                  O_BrakeProtectionAlarm => #AA_BrakeProtection,
                  O_SafetySwitchAlarm => #AA_SafetySwitch,
                  O_ConfigRampAlarm => #AC_ConfigRampAlm,
                  O_ConfigRampCalcAlarm => #AC_ConfigRampCalcAlm,
                  O_MotionStopWarning => #AD_MotionStop,
                  O_DriveFaultAlarm => #AB_Alarm,
                  O_DriveWarning => #AD_Warning,
                  O_Active => #MotorLoopActive,
                  O_DriveReady => #ReadyForOperation,
                  O_AlarmABCondition => #MotorLoopAlarmCond,
                  H_IAnim => #H_HMIMotor.H_IAnim);
   END_IF;
END_REGION

REGION Network 34: **** 7.3 - Submodule - Machine **** Motor loop Move UDT
   IF "TRUE" THEN #"H_GBLineConv-MDXPN-DFS22B".H_MotorIAnim[1].H_DWord := #H_HMIMotor.H_IAnim; END_IF;
END_REGION

REGION Network 35: **** 8 - Outputs **** Transfer OUT Transfer memory set
   // Transfer OUT Transfer memory set
   #O_TrfOutSetTM := #TrfOutSetTM;
END_REGION

REGION Network 36: **** 8 - Outputs **** Transfer OUT Ready To Deliver set
   // Transfer OUT Ready To Deliver set
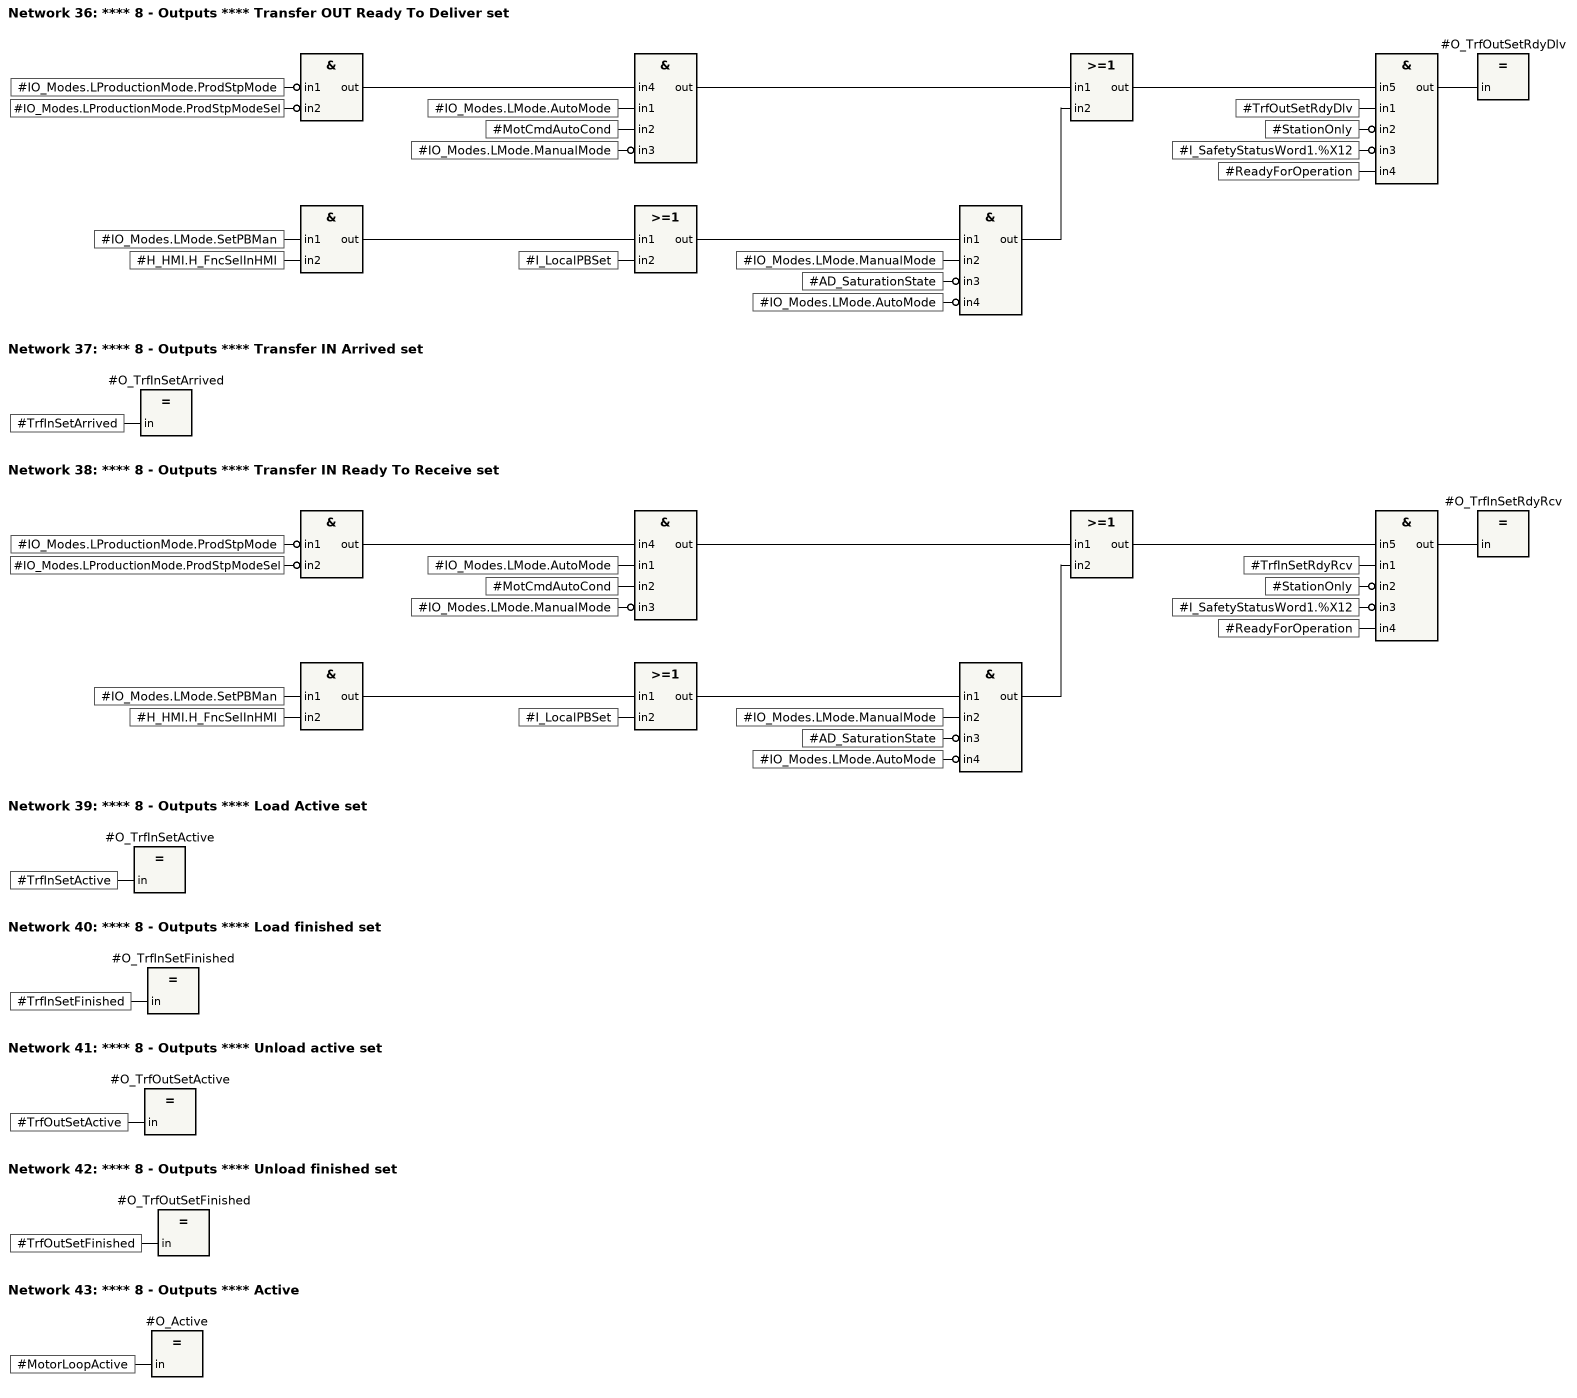
   #O_TrfOutSetRdyDlv := ((NOT #IO_Modes.LProductionMode.ProdStpMode AND NOT #IO_Modes.LProductionMode.ProdStpModeSel AND #IO_Modes.LMode.AutoMode AND #MotCmdAutoCond AND NOT #IO_Modes.LMode.ManualMode) OR (((#IO_Modes.LMode.SetPBMan AND #H_HMI.H_FncSelInHMI) OR #I_LocalPBSet) AND #IO_Modes.LMode.ManualMode AND NOT #AD_SaturationState AND NOT #IO_Modes.LMode.AutoMode)) AND #TrfOutSetRdyDlv AND NOT #StationOnly AND NOT #I_SafetyStatusWord1.%X12 AND #ReadyForOperation;
END_REGION

REGION Network 37: **** 8 - Outputs **** Transfer IN Arrived set
   // Transfer IN Arrived set
   #O_TrfInSetArrived := #TrfInSetArrived;
END_REGION

REGION Network 38: **** 8 - Outputs **** Transfer IN Ready To Receive set
   // Transfer IN Ready To Receive set
   #O_TrfInSetRdyRcv := ((NOT #IO_Modes.LProductionMode.ProdStpMode AND NOT #IO_Modes.LProductionMode.ProdStpModeSel AND #IO_Modes.LMode.AutoMode AND #MotCmdAutoCond AND NOT #IO_Modes.LMode.ManualMode) OR (((#IO_Modes.LMode.SetPBMan AND #H_HMI.H_FncSelInHMI) OR #I_LocalPBSet) AND #IO_Modes.LMode.ManualMode AND NOT #AD_SaturationState AND NOT #IO_Modes.LMode.AutoMode)) AND #TrfInSetRdyRcv AND NOT #StationOnly AND NOT #I_SafetyStatusWord1.%X12 AND #ReadyForOperation;
END_REGION

REGION Network 39: **** 8 - Outputs **** Load Active set
   // Load Active set
   #O_TrfInSetActive := #TrfInSetActive;
END_REGION

REGION Network 40: **** 8 - Outputs **** Load finished set
   // Load finished set
   #O_TrfInSetFinished := #TrfInSetFinished;
END_REGION

REGION Network 41: **** 8 - Outputs **** Unload active set
   // Unload active set
   #O_TrfOutSetActive := #TrfOutSetActive;
END_REGION

REGION Network 42: **** 8 - Outputs **** Unload finished set
   // Unload finished set
   #O_TrfOutSetFinished := #TrfOutSetFinished;
END_REGION

REGION Network 43: **** 8 - Outputs **** Active
   // motor active
   #O_Active := #MotorLoopActive;
END_REGION

REGION Network 44: **** 8 - Outputs **** Ready for operation
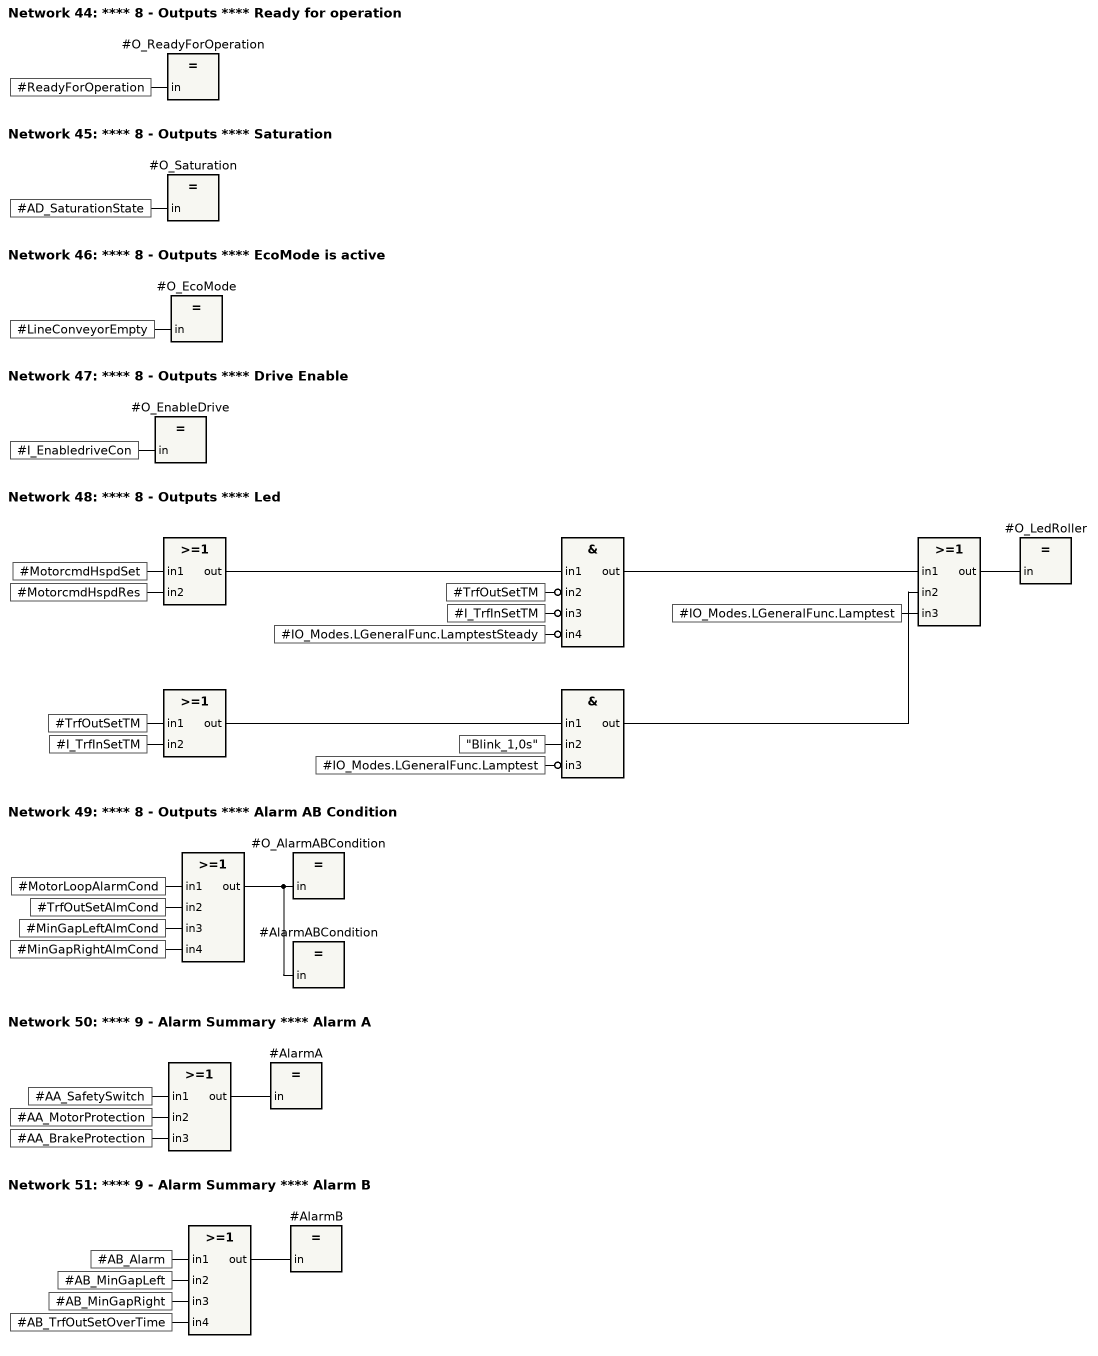
   #O_ReadyForOperation := #ReadyForOperation;
END_REGION

REGION Network 45: **** 8 - Outputs **** Saturation
   #O_Saturation := #AD_SaturationState;
END_REGION

REGION Network 46: **** 8 - Outputs **** EcoMode is active
   #O_EcoMode := #LineConveyorEmpty;
END_REGION

REGION Network 47: **** 8 - Outputs **** Drive Enable
   #O_EnableDrive := #I_EnabledriveCon;
END_REGION

REGION Network 48: **** 8 - Outputs **** Led
   // Led
   #O_LedRoller := ((#MotorcmdHspdSet OR #MotorcmdHspdRes) AND NOT #TrfOutSetTM AND NOT #I_TrfInSetTM AND NOT #IO_Modes.LGeneralFunc.LamptestSteady) OR ((#TrfOutSetTM OR #I_TrfInSetTM) AND "Blink_1,0s" AND NOT #IO_Modes.LGeneralFunc.Lamptest) OR #IO_Modes.LGeneralFunc.Lamptest;
END_REGION

REGION Network 49: **** 8 - Outputs **** Alarm AB Condition
   // Alarm AB Condition
   #O_AlarmABCondition := #MotorLoopAlarmCond OR #TrfOutSetAlmCond OR #MinGapLeftAlmCond OR #MinGapRightAlmCond;
   #AlarmABCondition := #O_AlarmABCondition;
END_REGION

REGION Network 50: **** 9 - Alarm Summary **** Alarm A
   // Alarm A
   #AlarmA := #AA_SafetySwitch OR #AA_MotorProtection OR #AA_BrakeProtection;
END_REGION

REGION Network 51: **** 9 - Alarm Summary **** Alarm B
   // Alarm B
   #AlarmB := #AB_Alarm OR #AB_MinGapLeft OR #AB_MinGapRight OR #AB_TrfOutSetOverTime;
END_REGION

REGION Network 52: **** 9 - Alarm Summary **** Alarm C
   // Alarm C
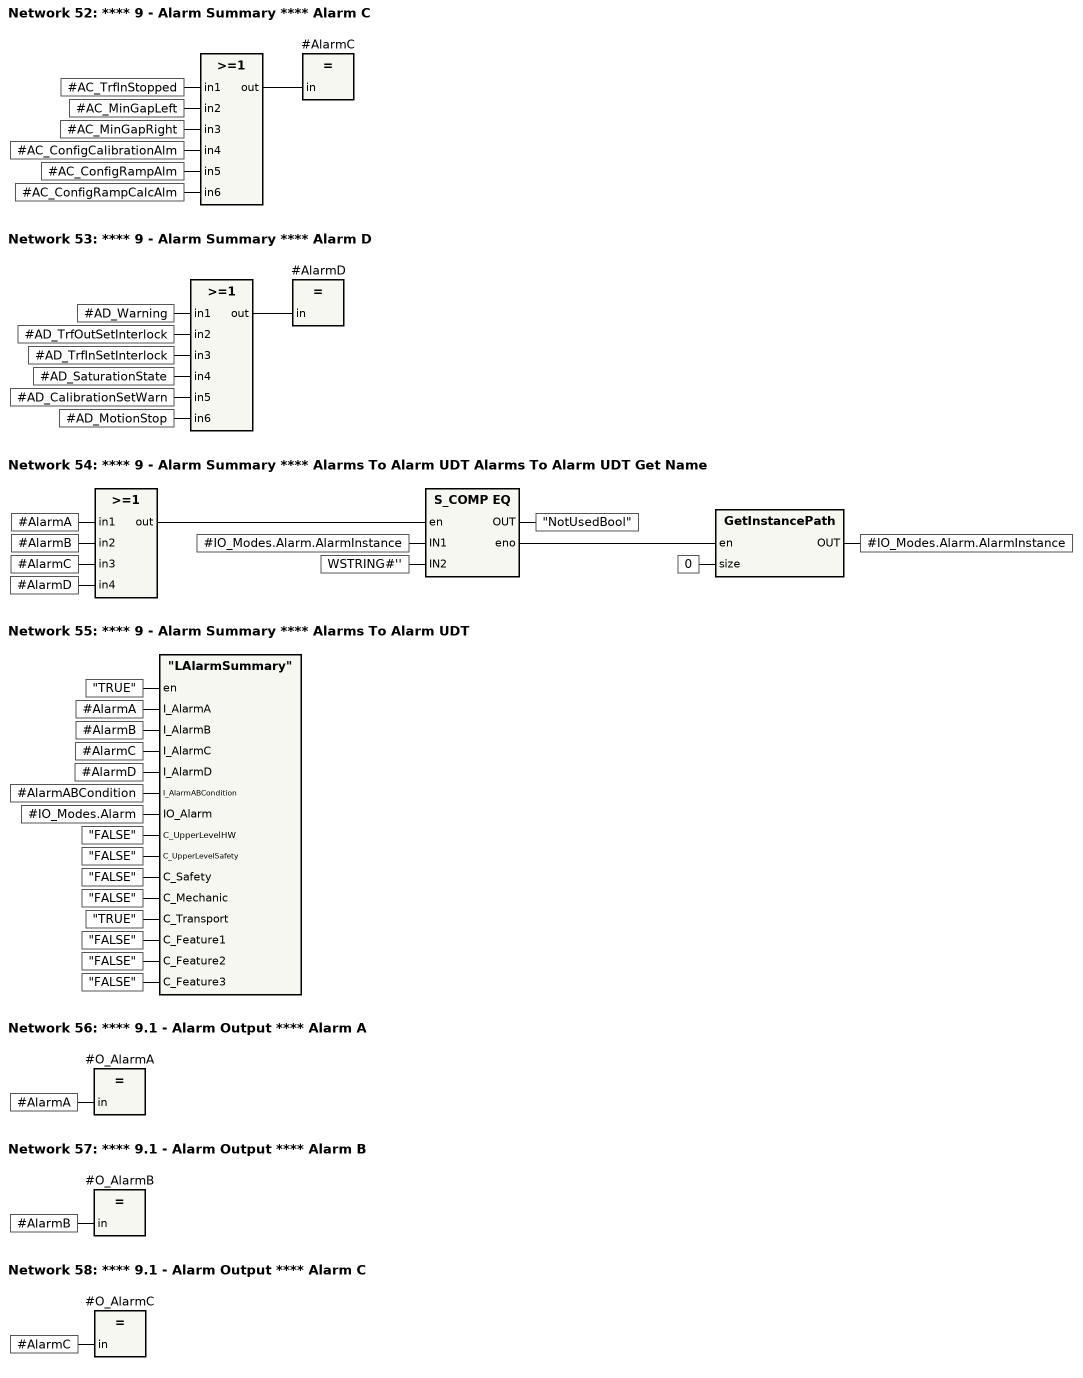
   #AlarmC := #AC_TrfInStopped OR #AC_MinGapLeft OR #AC_MinGapRight OR #AC_ConfigCalibrationAlm OR #AC_ConfigRampAlm OR #AC_ConfigRampCalcAlm;
END_REGION

REGION Network 53: **** 9 - Alarm Summary **** Alarm D
   // Alarm D
   #AlarmD := #AD_Warning OR #AD_TrfOutSetInterlock OR #AD_TrfInSetInterlock OR #AD_SaturationState OR #AD_CalibrationSetWarn OR #AD_MotionStop;
END_REGION

REGION Network 54: **** 9 - Alarm Summary **** Alarms To Alarm UDT Alarms To Alarm UDT Get Name
   // Alarm D
   S_COMP(EN := #AlarmA OR #AlarmB OR #AlarmC OR #AlarmD,
          IN1 := #IO_Modes.Alarm.AlarmInstance,
          IN2 := WSTRING#'',
          OUT => "NotUsedBool",
          ENO => #_w1);
   IF #_w1 THEN GetInstancePath(size := 0, OUT => #IO_Modes.Alarm.AlarmInstance); END_IF;
END_REGION

REGION Network 55: **** 9 - Alarm Summary **** Alarms To Alarm UDT
   // Alarm D
   IF "TRUE" THEN
       "LAlarmSummary"(I_AlarmA := #AlarmA,
                       I_AlarmB := #AlarmB,
                       I_AlarmC := #AlarmC,
                       I_AlarmD := #AlarmD,
                       I_AlarmABCondition := #AlarmABCondition,
                       IO_Alarm := #IO_Modes.Alarm,
                       C_UpperLevelHW := "FALSE",
                       C_UpperLevelSafety := "FALSE",
                       C_Safety := "FALSE",
                       C_Mechanic := "FALSE",
                       C_Transport := "TRUE",
                       C_Feature1 := "FALSE",
                       C_Feature2 := "FALSE",
                       C_Feature3 := "FALSE");
   END_IF;
END_REGION

REGION Network 56: **** 9.1 - Alarm Output **** Alarm A
   // Alarm A
   #O_AlarmA := #AlarmA;
END_REGION

REGION Network 57: **** 9.1 - Alarm Output **** Alarm B
   // Alarm B
   #O_AlarmB := #AlarmB;
END_REGION

REGION Network 58: **** 9.1 - Alarm Output **** Alarm C
   // Alarm C
   #O_AlarmC := #AlarmC;
END_REGION

REGION Network 59: **** 9.1 - Alarm Output **** Alarm D
   // Alarm D
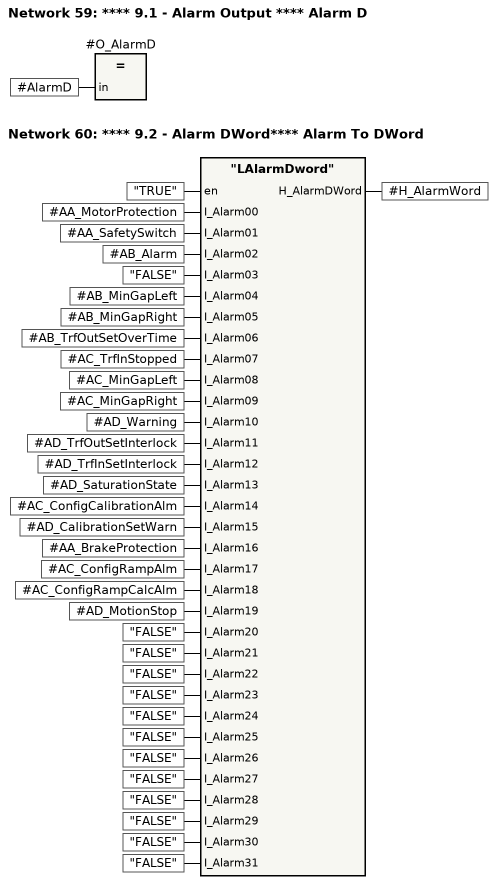
   #O_AlarmD := #AlarmD;
END_REGION

REGION Network 60: **** 9.2 - Alarm DWord**** Alarm To DWord
   // Alarm To Word
   IF "TRUE" THEN
       "LAlarmDword"(I_Alarm00 := #AA_MotorProtection,
                     I_Alarm01 := #AA_SafetySwitch,
                     I_Alarm02 := #AB_Alarm,
                     I_Alarm03 := "FALSE",
                     I_Alarm04 := #AB_MinGapLeft,
                     I_Alarm05 := #AB_MinGapRight,
                     I_Alarm06 := #AB_TrfOutSetOverTime,
                     I_Alarm07 := #AC_TrfInStopped,
                     I_Alarm08 := #AC_MinGapLeft,
                     I_Alarm09 := #AC_MinGapRight,
                     I_Alarm10 := #AD_Warning,
                     I_Alarm11 := #AD_TrfOutSetInterlock,
                     I_Alarm12 := #AD_TrfInSetInterlock,
                     I_Alarm13 := #AD_SaturationState,
                     I_Alarm14 := #AC_ConfigCalibrationAlm,
                     I_Alarm15 := #AD_CalibrationSetWarn,
                     I_Alarm16 := #AA_BrakeProtection,
                     I_Alarm17 := #AC_ConfigRampAlm,
                     I_Alarm18 := #AC_ConfigRampCalcAlm,
                     I_Alarm19 := #AD_MotionStop,
                     I_Alarm20 := "FALSE",
                     I_Alarm21 := "FALSE",
                     I_Alarm22 := "FALSE",
                     I_Alarm23 := "FALSE",
                     I_Alarm24 := "FALSE",
                     I_Alarm25 := "FALSE",
                     I_Alarm26 := "FALSE",
                     I_Alarm27 := "FALSE",
                     I_Alarm28 := "FALSE",
                     I_Alarm29 := "FALSE",
                     I_Alarm30 := "FALSE",
                     I_Alarm31 := "FALSE",
                     H_AlarmDWord => #H_AlarmWord);
   END_IF;
END_REGION
END_FUNCTION_BLOCK
